		fb_edit_mfps_bestuecken_b.st_config.b_config_fertig := FALSE;
		fb_edit_mfps_bestuecken_b.st_config.b_station_aktiv := TRUE;
		fb_edit_mfps_bestuecken_b.st_config.i16_meld_startindex := 860;
		fb_edit_mfps_bestuecken_b.st_config.str_beschreibung := ' ';
		fb_edit_mfps_bestuecken_b.st_config.str_instanz_name := 'Kurvenscheibeneditor Bestücken B-Achse';
		fb_edit_mfps_bestuecken_b.st_config.b_config_fertig := TRUE;

		fb_camtable_bestueckachse.st_config.b_config_fertig := FALSE;
		fb_camtable_bestueckachse.st_config.b_station_aktiv := TRUE;
		fb_camtable_bestueckachse.st_config.i16_meld_startindex := 880;
		fb_camtable_bestueckachse.st_config.str_beschreibung := ' ';
		fb_camtable_bestueckachse.st_config.str_instanz_name := 'Kurvenscheibeneditor Bestückachse';
		fb_camtable_bestueckachse.st_config.b_config_fertig := TRUE;

		(* Bestückbildgenerierung *)
		bbgen.st_config.b_config_fertig := FALSE;
		bbgen.st_config.b_station_aktiv := TRUE;
		bbgen.st_config.i16_meld_startindex := 700;
		bbgen.st_config.str_beschreibung := ' ';
		bbgen.st_config.str_instanz_name := 'Bestückbildgenerierung';
		bbgen.st_config.b_config_fertig := TRUE;
		
		(* Barcodereader *)
		barcode.fb.st_config.b_config_fertig := FALSE;
		barcode.fb.st_config.b_station_aktiv := TRUE;
		barcode.fb.st_config.i16_meld_startindex := 720;
		barcode.fb.st_config.str_beschreibung := ' ';
		barcode.fb.st_config.str_instanz_name := 'Barcodereader';
		barcode.fb.st_config.b_config_fertig := TRUE;
		
		(* Ballufftagreader *)
		balluff_tag_reader.fb.st_config.b_config_fertig := FALSE;
		balluff_tag_reader.fb.st_config.b_station_aktiv := TRUE;
		balluff_tag_reader.fb.st_config.i16_meld_startindex := 740;
		balluff_tag_reader.fb.st_config.str_beschreibung := ' ';
		balluff_tag_reader.fb.st_config.str_instanz_name := 'Ballufftagreader';
		balluff_tag_reader.fb.st_config.b_config_fertig := TRUE;

		(* WT-Transport Warteposition 1720 *)
		wt_transport_warteposition_1720.st_config.b_config_fertig := FALSE;
		wt_transport_warteposition_1720.st_config.i16_meld_startindex := 760;
		wt_transport_warteposition_1720.st_config.str_beschreibung := ' ';
		wt_transport_warteposition_1720.st_config.str_instanz_name := 'WT-Transport Warteposition 1720';
		wt_transport_warteposition_1720.st_config.b_config_fertig := TRUE;
		
		(* WT-Transport Beladestation 1720 *)
		wt_transport_beladen_1720.st_config.b_config_fertig := FALSE;
		wt_transport_beladen_1720.st_config.i16_meld_startindex := 780;
		wt_transport_beladen_1720.st_config.str_beschreibung := ' ';
		wt_transport_beladen_1720.st_config.str_instanz_name := 'WT-Transport Beladestation 1720';
		wt_transport_beladen_1720.st_config.b_config_fertig := TRUE;
		
		(* Rasterfolienmontge *)
		rasterfolienmontage.st_config.b_config_fertig := FALSE;
		rasterfolienmontage.st_config.b_station_aktiv := TRUE;
		rasterfolienmontage.st_config.i16_meld_startindex := 800;
		rasterfolienmontage.st_config.str_beschreibung := ' ';
		rasterfolienmontage.st_config.str_instanz_name := 'Rasterfolienmontge';
		rasterfolienmontage.st_config.b_config_fertig := TRUE;
		
		(* Rasterfolieneinzug *)
		rasterfolieneinzug.st_config.b_config_fertig := FALSE;
		rasterfolieneinzug.st_config.b_station_aktiv := TRUE;
		rasterfolieneinzug.st_config.i16_meld_startindex := 820;
		rasterfolieneinzug.st_config.str_beschreibung := ' ';
		rasterfolieneinzug.st_config.str_instanz_name := 'Rasterfolieneinzug';
		rasterfolieneinzug.st_config.b_config_fertig := TRUE;

		(*Tag lesen und schreiben *)
		Lesen_Schreiben_Tag.st_config.b_config_fertig := FALSE;
		Lesen_Schreiben_Tag.st_config.b_station_aktiv := TRUE;
		Lesen_Schreiben_Tag.st_config.i16_meld_startindex := 840;
		Lesen_Schreiben_Tag.st_config.str_beschreibung := ' ';
		Lesen_Schreiben_Tag.st_config.str_instanz_name := 'Tag lesen und schreiben';
		Lesen_Schreiben_Tag.st_config.b_config_fertig := TRUE;

		(* Wartung *)
		wartung.st_config.b_config_fertig := FALSE;
		wartung.st_config.b_station_aktiv := TRUE;
		wartung.st_config.i16_meld_startindex := 920;
		wartung.st_config.str_beschreibung := ' ';
		wartung.st_config.str_instanz_name := 'Wartung';
		wartung.st_config.b_config_fertig := TRUE;

		(*Service *)
		Service.st_config.b_config_fertig := FALSE;
		Service.st_config.b_station_aktiv := TRUE;
		Service.st_config.i16_meld_startindex := 900;
		Service.st_config.str_beschreibung := ' ';
		Service.st_config.str_instanz_name := 'Service';
		Service.st_config.b_config_fertig := TRUE;

		(*TouchProbe *)
		ST_TouchProbe.st_config.b_config_fertig := FALSE;
		ST_TouchProbe.st_config.b_station_aktiv := TRUE;
		ST_TouchProbe.st_config.i16_meld_startindex := 940;
		ST_TouchProbe.st_config.str_beschreibung := ' ';
		ST_TouchProbe.st_config.str_instanz_name := 'TouchProbe';
		ST_TouchProbe.st_config.b_config_fertig := TRUE;

		(*AutocheckinDaten *)
		ST_AutoCheckIn.fb_AutocheckinDaten.st_config.b_config_fertig:= FALSE;
		ST_AutoCheckIn.fb_AutocheckinDaten.st_config.b_station_aktiv:= TRUE;
		ST_AutoCheckIn.fb_AutocheckinDaten.st_config.i16_meld_startindex:=	960;
		ST_AutoCheckIn.fb_AutocheckinDaten.st_config.str_beschreibung:= ' ';
		ST_AutoCheckIn.fb_AutocheckinDaten.st_config.str_instanz_name:=	'AutoCheckInDaten';
		ST_AutoCheckIn.fb_AutocheckinDaten.st_config.b_config_fertig:= TRUE;

		(* WT-Transport Warteposition Achse 1700 *)
		wt_transport_warteposition_1700.st_config.b_config_fertig := FALSE;
		wt_transport_warteposition_1700.st_config.i16_meld_startindex := 400;
		wt_transport_warteposition_1700.st_config.str_beschreibung := ' ';
		wt_transport_warteposition_1700.st_config.str_instanz_name := 'WT-Transport Warteposition 1700';
		wt_transport_warteposition_1700.st_config.b_config_fertig := TRUE;
		
		(* WT-Transport Beladestation Achse 1700 *)
		wt_transport_beladen_achse_1700.st_config.b_config_fertig := FALSE;
		wt_transport_beladen_achse_1700.st_config.i16_meld_startindex := 420;
		wt_transport_beladen_achse_1700.st_config.str_beschreibung := ' ';
		wt_transport_beladen_achse_1700.st_config.str_instanz_name := 'WT-Transport Beladestation Achse 1700';
		wt_transport_beladen_achse_1700.st_config.b_config_fertig := TRUE;

		(* EtherCAT Diagnose *)
		Index:=1;
		EtherCatDiag[Index].st_config.b_config_fertig := FALSE;
		EtherCatDiag[Index].st_config.b_station_aktiv := TRUE;
		EtherCatDiag[Index].st_config.i16_meld_startindex := 980;
		EtherCatDiag[Index].st_config.str_beschreibung := ' ';
		EtherCatDiag[Index].st_config.str_instanz_name := 'Grundmaschine';
		EtherCatDiag[Index].st_config.b_config_fertig := TRUE;

		(* EtherCAT Diagnose *)
		Index:=2;
		EtherCatDiag[Index].st_config.b_config_fertig := FALSE;
		EtherCatDiag[Index].st_config.b_station_aktiv := TRUE;
		EtherCatDiag[Index].st_config.i16_meld_startindex := 985;
		EtherCatDiag[Index].st_config.str_beschreibung := ' ';
		EtherCatDiag[Index].st_config.str_instanz_name := 'Hublift links';
		EtherCatDiag[Index].st_config.b_config_fertig := TRUE;

		(* EtherCAT Diagnose *)
		Index:=3;
		EtherCatDiag[Index].st_config.b_config_fertig := FALSE;
		EtherCatDiag[Index].st_config.b_station_aktiv := TRUE;
		EtherCatDiag[Index].st_config.i16_meld_startindex := 990;
		EtherCatDiag[Index].st_config.str_beschreibung := ' ';
		EtherCatDiag[Index].st_config.str_instanz_name := 'Hublift rechts';
		EtherCatDiag[Index].st_config.b_config_fertig := TRUE;

		(* EtherCAT Diagnose *)
		Index:=4;
		EtherCatDiag[Index].st_config.b_config_fertig := FALSE;
		EtherCatDiag[Index].st_config.b_station_aktiv := TRUE;
		EtherCatDiag[Index].st_config.i16_meld_startindex := 995;
		EtherCatDiag[Index].st_config.str_beschreibung := ' ';
		EtherCatDiag[Index].st_config.str_instanz_name := 'Bandeinzug';
		EtherCatDiag[Index].st_config.b_config_fertig := TRUE;

		(* Melde-Arrays rücksetzen *)
		FOR i := 0 TO SIZEOF (garr_stoermeldungen) / SIZEOF (garr_stoermeldungen[0]) - 1 BY 1 DO
			garr_stoermeldungen[i] := 0;
		END_FOR
		FOR i := 0 TO SIZEOF (garr_betriebsmeldungen) / SIZEOF (garr_betriebsmeldungen[0]) - 1 BY 1 DO
			garr_betriebsmeldungen[i] := 0;
		END_FOR
ELSE
	b_config_fertig := TRUE;
END_IF

		
		
END_PROGRAM

(* POU Gemeinsamkeiten17xx/Achsen/ST_TouchProbe, ST *)
PROGRAM ST_TouchProbe
VAR_INPUT
	st_config						: struct_config;
	st_ctrl_in						: struct_ctrl_in;
END_VAR
VAR_OUTPUT
	st_ctrl_out					: struct_ctrl_out;
END_VAR
VAR
	fb_state_entry				: ST_StateEntry;
	st_ctrl_in_empty				: struct_ctrl_in;
	fb_ton_quitt					: TON;
	fb_ton_uez					: TON;
	fb_ton_wz					: TON;

	sm_CompareY				:BOOL;
	sm_CompareZ				:BOOL;
	sm_keinMessergebnisY		:BOOL;
	sm_keinMessergebnisZ		:BOOL;
	sm_WtAufSchlitten				:BOOL;

	i16_Counter					:INT;

	fb_TouchProbeLog			: FB_ExporString;	(* Fehlermeldungen in Errorlog (txt) schreiben *)
	s_FileName					: STRING;			(* Name Errorlogdatei *)
	s_ExportStr					: T_MaxString;		(* kompletter Text zum Eintrag in Errorlog *)
	s_ProductionsDate				: STRING;		(* Datum für Logeintrag *)

	lr_RecPosZ					:LREAL;		(*Wird beim Anlagenstart beschrieben*)
	lr_RecPosY					:LREAL;		(*Wird beim Anlagenstart beschrieben*)

END_VAR

VAR CONSTANT
	Trennzeichen					: STRING(3):=' |';
END_VAR
(*======================================================
   PRG: ST_TouchProbe
 ------------------------------------------------------
   Auth: 		Werner Friedl    						 
   Date: 		10.09.2019    						     
   Rev.: 		1.0	
   Desc:		Es werden nacheinander die Z- und Y Achse auf einen Messtaster gefahren und dabei
			die Ermittelten Tastpositionen in ein Lofile eingetregen. ("Projektpad"\TouchProbeLog)

			ACHTUNG!		auf dem Schlitten darf kein WT sein
							bei allen Anlagen Softwarelimits überprüfen und die Taster so motieren, dass sie kurz vor dem Softwarelimit schalten.

			Ablauf und Funktion.
			- bei einem Anlagen Neustart wird das erste Messergebnis in die VAR lr_RecPosZ und lr_RecPosY eingetragen.
			  Diese Messwerte werden dann mit allen darauf folgenden Messungen verglichen.
			- im Prg. "ST_AxisJobCtrl_Motion" muss die Touchprobe Funktion eingefügt sein ( MOVE_TOUCH_PROBE)

			gst_datensatz.st_md.lr_ToleranzTouchProbe				(Toleranz für den Vergleich)
			gst_datensatz.st_md.i16_WdhTouchProbe				(Anzahl der WT-wechsel bis zur nächsten Messung bei 0 wird keine Prüfung gemacht)

			Das Programm wird im ST_WT_Transport_Beladen gestartet (Schritt 140)

   Historie:   1.0

 ========================================================*)
(* Zeiten *)
fb_ton_wz(IN:= , PT:= , Q=>  , ET=> );
fb_ton_uez(IN:= , PT:= , Q=>  , ET=> );
fb_ton_quitt(IN:= , PT:= t#100ms, Q=> , ET=> );

(* Flanken *)

(* Toplevel *)
IF fb_state_entry.i16_next_step > INIT AND fb_state_entry.i16_next_step < FEHLER THEN
	IF fb_state_entry.i16_next_step < STOP THEN
		IF st_ctrl_in.b_stop THEN
			fb_state_entry.i16_next_step := STOP;
		END_IF
	END_IF

	IF	axis_y_achse.st_ctrl.out.b_fehler	OR
		axis_z_achse.st_ctrl.out.b_fehler OR
		NOT ST_Safetyprogramm.se_steuerung_ein THEN
		fb_state_entry.i16_next_step := FEHLER;
	END_IF

END_IF

(* ==================================Schrittkette================================ *)
fb_state_entry(i16_pos:= 1);

CASE fb_state_entry.i16_step OF
(*=======================================================*)
INIT_OBJ:
	IF st_config.b_config_fertig THEN
		fb_state_entry.i16_next_step := INIT;
	END_IF

(*=======================================================*)
INIT:
	IF fb_state_entry.E THEN
		fb_ton_wz.IN := FALSE;
		fb_ton_uez.IN	:= FALSE;
		fb_ton_quitt.IN := FALSE;

		sm_CompareY:=FALSE;
		sm_CompareZ:=FALSE;
		sm_keinMessergebnisY:=FALSE;
		sm_keinMessergebnisZ:=FALSE;
		sm_WtAufSchlitten:=	FALSE;
	END_IF

	(*-----------------------Weiterschaltbedingungen----------------------------*)
	IF 	st_ctrl_in.b_init THEN
		fb_state_entry.i16_next_step := 20;
	END_IF

(*=======================================================*)
20: (* Initialisierung*)

	(*-----------------------Weiterschaltbedingungen----------------------------*)
	fb_state_entry.i16_next_step := BEREIT;

(*=======================================================*)
BEREIT:	(* Warte auf Anforderung von vorheriger Station zum aufnehmen des WT *)
	IF 	fb_state_entry.E THEN
		st_ctrl_out.b_bereit := TRUE;
	END_IF

	(*-----------------------Weiterschaltbedingungen----------------------------*)
	IF 	st_ctrl_in.b_start  OR st_ctrl_in.b_start_2 THEN
		fb_state_entry.i16_next_step := 110;
	END_IF

	IF 	fb_state_entry.X THEN
		st_ctrl_out.b_fertig := FALSE;
		st_ctrl_out.b_busy := TRUE;
	END_IF

(*=======================================================*)
110: (* Prüfe Startbedinung*)

	(*-----------------------Weiterschaltbedingungen----------------------------*)
	(*Prüfen ob ein Taster angeklemmt ist*)
	IF	NOT ST_Z_Achse.fb_axis.b_TriggerInput OR
		gst_datensatz.st_md.i16_WdhTouchProbe <= 0 OR
		gst_datensatz.st_md.lr_ToleranzTouchProbe <= 0 THEN
		fb_state_entry.i16_next_step := BEREIT;
		st_ctrl_out.b_fertig := TRUE;
		st_ctrl_out.b_busy := FALSE;
	ELSE
		IF	i16_Counter >= gst_datensatz.st_md.i16_WdhTouchProbe  OR
			i16_Counter = 0 THEN
			fb_state_entry.i16_next_step := 115;
		ELSE
			st_ctrl_out.b_fertig := TRUE;
			st_ctrl_out.b_busy := FALSE;
			fb_state_entry.i16_next_step := BEREIT;
		END_IF
	END_IF

	IF 	fb_state_entry.X THEN
		i16_Counter:=i16_Counter+1;
	END_IF

(*=======================================================*)
115: (* Prüfe ob Schlitten ohne WT ist*)
	IF fb_state_entry.E THEN
		fb_ton_wz.PT := t#1000ms;
	END_IF

	IF	gst_datensatz.st_md.i16_typ_zelle = BESTUECKZELLE_1720   THEN
		fb_ton_wz.IN:=ST_WT_Transport_Beladen_1720.e_wt_auf_beladepos;
		IF NOT ST_WT_Transport_Beladen_1720.e_wt_auf_beladepos THEN
			fb_state_entry.i16_next_step := 120;
		END_IF
	ELSE
		fb_ton_wz.IN:=ST_WT_Transport_Beladen.e_wt_auf_beladepos;
		IF NOT ST_WT_Transport_Beladen.e_wt_auf_beladepos THEN
			fb_state_entry.i16_next_step := 120;
		END_IF
	END_IF

	IF	fb_ton_wz.Q THEN
		sm_WtAufSchlitten:=TRUE;
		fb_state_entry.i16_next_step := FEHLER;
	END_IF

	IF fb_state_entry.X THEN
		fb_ton_wz.IN := FALSE;
	END_IF

(*=======================================================*)
120: (* CAM_OUT_SLAVE*)
	IF fb_state_entry.E THEN
		ST_Z_Achse.b_start_in := TRUE;
	END_IF

	(*-----------------------Weiterschaltbedingungen----------------------------*)
	IF	axis_z_achse.st_ctrl.out.b_busy  THEN
		fb_state_entry.i16_next_step := 122;
	END_IF

(*=======================================================*)
122:(*warten auf  fertig*)
	(*-----------------------Weiterschaltbedingungen----------------------------*)
	IF	axis_z_achse.st_ctrl.out.b_fertig  THEN
		fb_state_entry.i16_next_step := 124;
	END_IF

(*=======================================================*)
124:(*prüfe CoupleState*)

	IF 	(y_achse.NcToPlc.CoupleState = 0 OR gst_datensatz.st_md.i16_typ_zelle = BESTUECKZELLE_1720)AND
	 	z_achse.NcToPlc.CoupleState = 0  THEN
		fb_state_entry.i16_next_step := 126;
	END_IF

(*=======================================================*)
126: (* Z-Achse vor TouchProbe fahren*)
	IF fb_state_entry.E THEN
		ST_Z_Achse.lr_Achspos_in:=-95 + 20 ;				(*Taster befindet sich in Der Nähe vom Motor*)
		ST_Z_Achse.lr_Velo_in:=ST_Z_Achse.st_geschwindigkeiten.lr_auto_max ;
		ST_Z_Achse.enu_cmd_in:=MOVE_TOUCH_PROBE;
		ST_Z_Achse.b_start_in := TRUE;
	END_IF

	(*-----------------------Weiterschaltbedingungen----------------------------*)
	IF	axis_z_achse.st_ctrl.out.b_busy  THEN
		fb_state_entry.i16_next_step := 128;
	END_IF

(*=======================================================*)
128:(*warten auf  fertig*)
	(*-----------------------Weiterschaltbedingungen----------------------------*)
	IF	axis_z_achse.st_ctrl.out.b_fertig  THEN
		fb_state_entry.i16_next_step := 130;
	END_IF

(*=======================================================*)
130: (* Z-Achse auf TouchProbe fahren*)
	IF fb_state_entry.E THEN
		ST_Z_Achse.lr_Achspos_in:=-95 ;				(*Taster befindet sich in Der Nähe vom Motor*)
		ST_Z_Achse.lr_Velo_in:=ST_Z_Achse.st_geschwindigkeiten.lr_auto_max / 5;
		ST_Z_Achse.enu_cmd_in:=MOVE_TOUCH_PROBE;
		ST_Z_Achse.b_start_in := TRUE;
	END_IF

	(*-----------------------Weiterschaltbedingungen----------------------------*)
	IF	axis_z_achse.st_ctrl.out.b_busy  THEN
		fb_state_entry.i16_next_step := 132;
	END_IF

(*=======================================================*)
132:(*warten auf  fertig*)
	(*-----------------------Weiterschaltbedingungen----------------------------*)
	IF	axis_z_achse.st_ctrl.out.b_fertig  THEN
		fb_state_entry.i16_next_step := 134;
	END_IF

(*=======================================================*)
134: (* Z-Achse vom TouchProbe runter fahren und Positionieren für die Y Achse *)
	IF fb_state_entry.E THEN
		IF	gst_datensatz.st_md.i16_typ_zelle <> BESTUECKZELLE_1720 THEN
			ST_Z_Achse.lr_Achspos_in:=70;				(*Taster befindet sich in DerNähe vom Motor*)
		ELSE
			ST_Z_Achse.lr_Achspos_in:=gst_datensatz.st_md.st_md_z_achse.lr_wt_uebergabepos  ;
		END_IF
		ST_Z_Achse.lr_Velo_in:=ST_Z_Achse.st_geschwindigkeiten.lr_auto_max ;
		ST_Z_Achse.enu_cmd_in:=MOVE_ABSOLUTE;
		ST_Z_Achse.b_start_in := TRUE;
	END_IF

	(*-----------------------Weiterschaltbedingungen----------------------------*)
	IF	axis_z_achse.st_ctrl.out.b_busy  THEN
		fb_state_entry.i16_next_step := 140;
	END_IF

(*=======================================================*)
140:(*warten auf  fertig*)
	(*-----------------------Weiterschaltbedingungen----------------------------*)
	IF	axis_z_achse.st_ctrl.out.b_fertig  THEN

		IF	gst_datensatz.st_md.i16_typ_zelle = BESTUECKZELLE_1720 THEN
			fb_state_entry.i16_next_step := 220;
		ELSE
			fb_state_entry.i16_next_step := 150;
		END_IF
	END_IF

(*=======================================================*)
150: (* Y-Achse auf TouchProbe fahren*)
	IF fb_state_entry.E THEN
		ST_Y_Achse.lr_Achspos_in:=30;				(*Taster befindet sich in der Nähe vom Motor*)
		ST_Y_Achse.lr_Velo_in:=ST_Y_Achse.st_geschwindigkeiten.lr_auto_max;
		ST_Y_Achse.enu_cmd_in:=MOVE_ABSOLUTE;
		ST_Y_Achse.b_start_in := TRUE;
	END_IF

	(*-----------------------Weiterschaltbedingungen----------------------------*)
	IF	axis_y_achse.st_ctrl.out.b_busy  THEN
		fb_state_entry.i16_next_step := 160;
	END_IF

(*=======================================================*)
160:(*warten auf  fertig*)
	(*-----------------------Weiterschaltbedingungen----------------------------*)
	IF	axis_y_achse.st_ctrl.out.b_fertig  THEN
		fb_state_entry.i16_next_step := 162;
	END_IF

(*=======================================================*)
162: (* Y-Achse auf TouchProbe fahren*)
	IF fb_state_entry.E THEN
		ST_Y_Achse.lr_Achspos_in:=65;				(*Taster befindet sich in der Nähe vom Motor*)
		ST_Y_Achse.lr_Velo_in:=ST_Y_Achse.st_geschwindigkeiten.lr_auto_max / 5;
		ST_Y_Achse.enu_cmd_in:=MOVE_TOUCH_PROBE;
		ST_Y_Achse.b_start_in := TRUE;
	END_IF

	(*-----------------------Weiterschaltbedingungen----------------------------*)
	IF	axis_y_achse.st_ctrl.out.b_busy  THEN
		fb_state_entry.i16_next_step := 164;
	END_IF

(*=======================================================*)
164:(*warten auf  fertig*)
	(*-----------------------Weiterschaltbedingungen----------------------------*)
	IF	axis_y_achse.st_ctrl.out.b_fertig  THEN
		fb_state_entry.i16_next_step := 170;
	END_IF

(*=======================================================*)
170: (* Y-Achse vom TouchProbe runter fahren*)
	IF fb_state_entry.E THEN
		ST_Y_Achse.lr_Achspos_in:=30 ;
		ST_Y_Achse.lr_Velo_in:=ST_Y_Achse.st_geschwindigkeiten.lr_auto_max;
		ST_Y_Achse.enu_cmd_in:=MOVE_ABSOLUTE;
		ST_Y_Achse.b_start_in := TRUE;
	END_IF

	(*-----------------------Weiterschaltbedingungen----------------------------*)
	IF	axis_y_achse.st_ctrl.out.b_busy  THEN
		fb_state_entry.i16_next_step := 180;
	END_IF

(*=======================================================*)
180:(*warten auf  Vorschub zurück fertig*)
	(*-----------------------Weiterschaltbedingungen----------------------------*)
	IF	axis_y_achse.st_ctrl.out.b_fertig  THEN
		fb_state_entry.i16_next_step := 190;
	END_IF

(*=======================================================*)
190: (* Y-Achse vom TouchProbe runter fahren*)
	IF fb_state_entry.E THEN
		ST_Y_Achse.lr_Achspos_in:=gst_datensatz.st_md.st_md_y_achse.lr_wt_uebergabepos;
		ST_Y_Achse.enu_cmd_in:=MOVE_ABSOLUTE;
		ST_Y_Achse.b_start_in := TRUE;
		ST_Z_Achse.lr_Achspos_in:=gst_datensatz.st_md.st_md_z_achse.lr_wt_uebergabepos  ;
		ST_Z_Achse.enu_cmd_in:=MOVE_ABSOLUTE;
		ST_Z_Achse.b_start_in := TRUE;
	END_IF

	(*-----------------------Weiterschaltbedingungen----------------------------*)
	IF	axis_y_achse.st_ctrl.out.b_busy  AND
		axis_z_achse.st_ctrl.out.b_busy THEN
		fb_state_entry.i16_next_step := 200;
	END_IF

(*=======================================================*)
200:(*warten auf  Vorschub zurück fertig*)
	(*-----------------------Weiterschaltbedingungen----------------------------*)
	IF	axis_y_achse.st_ctrl.out.b_fertig AND
		axis_z_achse.st_ctrl.out.b_fertig THEN
		fb_state_entry.i16_next_step := 210;
	END_IF

(*=======================================================*)
210: (* Y- und Z_Achse auf Startposition fahren*)
	IF fb_state_entry.E THEN
		ST_Z_Achse.enu_cmd_in:=CAM_IN_SLAVE;			(*Y-Achse wird wieder angekoppelt*)
		ST_Z_Achse.b_start_in := TRUE;
	END_IF

	(*-----------------------Weiterschaltbedingungen----------------------------*)
	IF	axis_z_achse.st_ctrl.out.b_busy THEN
		fb_state_entry.i16_next_step := 220;
	END_IF

(*=======================================================*)
220:(*warten auf  Vorschub zurück fertig*)
	(*-----------------------Weiterschaltbedingungen----------------------------*)
	IF	axis_z_achse.st_ctrl.out.b_fertig  THEN
		fb_state_entry.i16_next_step := 230;
		st_ctrl_out.b_fertig := TRUE;
		st_ctrl_out.b_busy := FALSE;
	END_IF

(*=======================================================*)
230:(*Wenn die RecPos=0 sind dann funktionieren die Messtaster nicht*)

	IF	gst_datensatz.st_md.i16_typ_zelle <> BESTUECKZELLE_1720 THEN
		sm_keinMessergebnisY := ST_Y_Achse.lr_RecPos = 0;
	END_IF
	sm_keinMessergebnisZ := ST_Z_Achse.lr_RecPos = 0;

	(*-----------------------Weiterschaltbedingungen----------------------------*)
	IF	sm_keinMessergebnisY OR
		sm_keinMessergebnisZ THEN
		fb_state_entry.i16_next_step := FEHLER;
	ELSE
		fb_state_entry.i16_next_step := 500;
		i16_Counter:=1;
	END_IF

(*=======================================================*)
500:	(*Eintrag in die ErrorLog===========================================*)
	IF	fb_state_entry.E THEN

		s_ProductionsDate:=DT_TO_SPECIALSTRING_YYYY_MM(inDT:=gdt_system_time);
		s_FileName:=CONCAT('TouchProbeLog_',s_ProductionsDate);
		s_FileName:=CONCAT(s_FileName,'.txt');
		s_ExportStr:=DELETE(DT_TO_STRING(gdt_system_time),3,1);
		s_ExportStr:=CONCAT(s_ExportStr,Trennzeichen);
		s_ExportStr:=CONCAT(s_ExportStr,'Axis Z: ');
		s_ExportStr:=CONCAT(s_ExportStr,LREAL_TO_FMTSTR(ST_Z_Achse.lr_RecPos,5,TRUE));
		IF	gst_datensatz.st_md.i16_typ_zelle <> BESTUECKZELLE_1720 THEN
			s_ExportStr:=CONCAT(s_ExportStr,Trennzeichen);
			s_ExportStr:=CONCAT(s_ExportStr,'Axis Y: ');
			s_ExportStr:=CONCAT(s_ExportStr,LREAL_TO_FMTSTR(ST_Y_Achse.lr_RecPos,5,TRUE));
		END_IF

		IF 	lr_RecPosY = 0 THEN		(*Wird beim Anlagenstart beschrieben*)
			lr_RecPosY:= ST_Y_Achse.lr_RecPos;
		END_IF

		IF 	lr_RecPosZ = 0 THEN		(*Wird beim Anlagenstart beschrieben*)
			lr_RecPosZ:= ST_Z_Achse.lr_RecPos;
			s_ExportStr:=CONCAT(s_ExportStr,' start compare ');
		END_IF

		sm_CompareY:=ABS(lr_RecPosY - ST_Y_Achse.lr_RecPos) > gst_datensatz.st_md.lr_ToleranzTouchProbe;
		sm_CompareZ:=ABS(lr_RecPosZ - ST_Z_Achse.lr_RecPos) > gst_datensatz.st_md.lr_ToleranzTouchProbe;

		IF 	sm_CompareY OR
			sm_CompareZ THEN
			s_ExportStr:=CONCAT(s_ExportStr,' error compare   difference > ');
			s_ExportStr:=CONCAT(s_ExportStr,LREAL_TO_FMTSTR(gst_datensatz.st_md.lr_ToleranzTouchProbe,4,TRUE));
		END_IF

	END_IF

	(*-----------------------Weiterschaltbedingungen----------------------------*)
	IF	NOT fb_TouchProbeLog.Busy AND
		NOT fb_TouchProbeLog.Error  THEN
		fb_state_entry.i16_next_step:=510;
	ELSE
		fb_state_entry.i16_next_step:=FEHLER;
	END_IF

(*=======================================================*)
510:	(* Starte Schreibvorgang *)
	IF	fb_state_entry.E THEN
		fb_TouchProbeLog.Start:=TRUE;
	END_IF

	(*-----------------------Weiterschaltbedingungen----------------------------*)
	IF	NOT fb_TouchProbeLog.Busy AND
		fb_TouchProbeLog.Done THEN
		fb_state_entry.i16_next_step:=BEREIT;
	END_IF
	IF	fb_TouchProbeLog.Error OR
		sm_CompareY OR
 		sm_CompareZ THEN
		fb_state_entry.i16_next_step:=FEHLER;
	END_IF


(*=======================================================*)
FEHLER:
	IF fb_state_entry.E THEN
		fb_ton_quitt.IN := FALSE;
		st_ctrl_out.b_fehler := TRUE;
		st_ctrl_out.b_bereit := FALSE;
		st_ctrl_out.b_fertig := FALSE;
		st_ctrl_out.b_busy := FALSE;
	END_IF

	(*-----------------------Weiterschaltbedingungen----------------------------*)
	IF st_ctrl_in.b_quitt AND NOT fb_state_entry.E THEN
		st_ctrl_out.b_fehler := FALSE;
		fb_ton_quitt.IN := TRUE;
	END_IF


	IF fb_ton_quitt.Q THEN
		fb_ton_quitt.IN := FALSE;
		fb_state_entry.i16_next_step := INIT;
	END_IF

(*=======================================================*)
STOP:
	IF fb_state_entry.E THEN
		fb_ton_quitt.IN := FALSE;
		st_ctrl_out.b_gestoppt := TRUE;
		st_ctrl_out.b_bereit := FALSE;
		st_ctrl_out.b_fertig := FALSE;
		st_ctrl_out.b_busy := FALSE;
	END_IF

	(*-----------------------Weiterschaltbedingungen----------------------------*)
	IF 	st_ctrl_in.b_quitt AND NOT fb_state_entry.E THEN
		st_ctrl_out.b_gestoppt := FALSE;
		fb_ton_quitt.IN := TRUE;
	END_IF

	IF fb_ton_quitt.Q THEN
		fb_ton_quitt.IN := FALSE;
		fb_state_entry.i16_next_step := INIT;
	END_IF
END_CASE

st_ctrl_in:=st_ctrl_in_empty;

fb_state_entry(i16_pos:= 2);

IF st_config.b_config_fertig THEN
	(* Fehlermeldungen und Betriebsmeldungen ab dem Startindex in die globalen Meldungsarrays schreiben *)
	garr_stoermeldungen[st_config.i16_meld_startindex + 0] := sm_CompareY;
	garr_stoermeldungen[st_config.i16_meld_startindex + 1] := sm_CompareZ;
	garr_stoermeldungen[st_config.i16_meld_startindex + 2] := sm_keinMessergebnisY;
	garr_stoermeldungen[st_config.i16_meld_startindex + 3] := sm_keinMessergebnisZ;
	garr_stoermeldungen[st_config.i16_meld_startindex + 4] := sm_WtAufSchlitten;
	garr_stoermeldungen[st_config.i16_meld_startindex + 5] := FALSE;
	garr_stoermeldungen[st_config.i16_meld_startindex + 6] := FALSE;
	garr_stoermeldungen[st_config.i16_meld_startindex + 7] := FALSE;
	garr_stoermeldungen[st_config.i16_meld_startindex + 8] := FALSE;
	garr_stoermeldungen[st_config.i16_meld_startindex + 9] := FALSE;

	garr_betriebsmeldungen[st_config.i16_meld_startindex + 0] := FALSE;
	garr_betriebsmeldungen[st_config.i16_meld_startindex + 1] := FALSE;
	garr_betriebsmeldungen[st_config.i16_meld_startindex + 2] := FALSE;
	garr_betriebsmeldungen[st_config.i16_meld_startindex + 3] := FALSE;
	garr_betriebsmeldungen[st_config.i16_meld_startindex + 4] := FALSE;
	garr_betriebsmeldungen[st_config.i16_meld_startindex + 5] := FALSE;
	garr_betriebsmeldungen[st_config.i16_meld_startindex + 6] := FALSE;
	garr_betriebsmeldungen[st_config.i16_meld_startindex + 7] := FALSE;
	garr_betriebsmeldungen[st_config.i16_meld_startindex + 8] := FALSE;
	garr_betriebsmeldungen[st_config.i16_meld_startindex + 9] := FALSE;

END_IF


fb_TouchProbeLog(
	Start:= ,
	Reset:= ,
	ExportStr:= s_ExportStr,
	FileName:= s_FileName,
	Path:=  CONCAT(s_Projekt_path,'TouchProbeLog\'),
	Mode:=FOPEN_MODEAPPEND,	(*am Ende anhängen*)
	Ready=> ,
	Busy=> ,
	Done=> ,
	Error=> ,
	ErrorMsg=> );
END_PROGRAM

(* POU EPT Lib/Daten/FB_ExporString, ST *)
FUNCTION_BLOCK FB_ExporString
VAR_INPUT
	Start				:BOOL;
	Reset			:BOOL;
	ExportStr			:STRING(255);
	FileName		:STRING(255);
	Path				:STRING(255);
	Mode			:DWORD;
END_VAR
VAR_OUTPUT
	Ready				:BOOL;
	Busy				:BOOL;
	Done				:BOOL;
	Error				:BOOL;
	ErrorMsg			:STRING(255);

END_VAR
VAR
	fb_state_entry		:ST_StateEntry;
	nErrId				:UDINT;
	i					:UINT;

	fbFileOpen			:FB_FileOpen;
	fbFilePuts			:FB_FilePuts;
	fbFileClose			:FB_FileClose;

	hFile				:UINT;

	ProductionDate		:STRING;

END_VAR

VAR CONSTANT
	Zeilenumbruch		:STRING:='$R$N';
END_VAR
(*======================================================
   PRG: FB_ExportString
 ------------------------------------------------------
   Auth: 		Werner Friedl    						 
   Date: 		30.10.2014    						     
   Rev.: 		1.0	
   Desc:		
		
   Historie:   1.0

 ========================================================*)
fb_state_entry(i16_pos:= 1);

CASE fb_state_entry.i16_step OF

0:	(*Objekt initialisieren*)
	fb_state_entry.i16_next_step:=INIT;

10:	(*initialisieren*)
	fb_state_entry.i16_next_step:=BEREIT;

BEREIT:(*Start*)

	IF	Start THEN  (*initialisieren*)
		Start:=FALSE;
		Busy:=TRUE;
		Error:=FALSE;
		Done:=FALSE;
		nErrId:=0;
		ErrorMsg:='';
		fb_state_entry.i16_next_step:=110;

	END_IF

110: (*Datei erstellen*)

	FileName:=CONCAT(Path,FileName);

	fbFileOpen.sPathName:=FileName;
 	fbFileOpen.bExecute:=TRUE;

	IF 	NOT fbFileOpen.bBusy   THEN
		fb_state_entry.i16_next_step:=120;
	END_IF

120: (*Datei erstellen*)

	IF 	NOT fbFileOpen.bBusy THEN
		fbFileOpen.bExecute:=FALSE;
		IF 	fbFileOpen.bError THEN
			nErrId:=fbFileOpen.nErrId;
			fb_state_entry.i16_next_step:=FEHLER;
			ErrorMsg:='Fehler beim Öffnen der Datei';
		ELSE
			fb_state_entry.i16_next_step:=130;
		END_IF
	END_IF

130: (*String in Datei eintragen*)
	IF fb_state_entry.E THEN
		;
	END_IF

	fbFilePuts.sLine:=CONCAT(ExportStr,Zeilenumbruch);
	fbFilePuts.bExecute:=TRUE;

	IF  fbFilePuts.bBusy THEN
		fb_state_entry.i16_next_step:=140;
	END_IF

140: (*String in Datei eintragen*)

	IF 	NOT fbFilePuts.bBusy THEN
		fbFilePuts.bExecute:=FALSE;
		IF 	fbFilePuts.bError THEN
			nErrId:=fbFilePuts.nErrId;
			fb_state_entry.i16_next_step:=150;
			ErrorMsg:='Fehler beim String Eintragen in der Datei';
			Error:=TRUE;
		ELSE
			fb_state_entry.i16_next_step:=150;
		END_IF
	END_IF

150:(*Datei schließen*)

	fbFileClose.bExecute:=TRUE;
	IF 	fbFileClose.bBusy THEN
		fb_state_entry.i16_next_step:=160;
	END_IF

160:(*Datei schließen*)

	IF NOT fbFileClose.bBusy THEN
		fbFileClose.bExecute:=FALSE;
		IF 	fbFileClose.bError THEN
			nErrId:=fbFileClose.nErrId;
			ErrorMsg:='Fehler beim Schließen der Datei';
			Error:=TRUE;
		ELSE
			fb_state_entry.i16_next_step:=170;
		END_IF
	END_IF

	IF	Error THEN
		fb_state_entry.i16_next_step:=FEHLER;
	END_IF

170: (*fertig*)
	Busy:=FALSE;
	Done:=TRUE;
	fb_state_entry.i16_next_step:=10;

FEHLER: (*Fehler*)
	fb_state_entry.i16_next_step:=10;
	Busy:=FALSE;
	Error:=TRUE;
END_CASE

fb_state_entry(i16_pos:= 2 );

fbFileOpen(
	sNetId:='',
	sPathName:= ,
	nMode:=mode,
	ePath:=PATH_GENERIC,
	bExecute:= ,
	tTimeout:=T#1s,
	hFile=> hFile);

fbFilePuts(
	sNetId:='',
	hFile:=hFile,
	sLine:= ,
	bExecute:= ,
	tTimeout:=t#1s);

fbFileClose(
	sNetId:='',
	hFile:=hFile,
	bExecute:= ,
	tTimeout:=t#1s);
END_FUNCTION_BLOCK

(* POU Maschine1720/WT Transport/ST_WT_Transport_Beladen_1720, ST *)
PROGRAM ST_WT_Transport_Beladen_1720
VAR_INPUT
	st_config								: struct_config;
	st_ctrl_in								: struct_ctrl_in;
END_VAR
VAR_IN_OUT
	st_visu								: struct_visu;
END_VAR
VAR_OUTPUT
	st_ctrl_out							: struct_ctrl_out;
	t_WT_WechselZeit					: TIME := t#0ms;
	t_traegerwechselzeit					: TIME := t#0ms;
	t_Zentrierer_ausfahren					: TIME := t#0ms;
	t_Zentrierer_einfahren					: TIME := t#0ms;
	t_komplett_zyklus						: TIME := t#0ms;
END_VAR
VAR
	fb_ton_uez							: TON;
	fb_ton_wz							: TON;
	fb_ton_quitt							: TON;
	fb_ton_wt_auf_beladepos				: TON;
	fb_tof_wt_auf_beladepos				: TOF;
	fb_r_trig_start							: R_TRIG;
	fb_r_trig_beladepos					: R_TRIG;
	fb_r_trig_beladepos_verlassen			: R_TRIG;
	fb_state_entry							: ST_StateEntry;
	fb_traegerwechselzeit					: ST_Taktzeit;
	fb_WT_WechselZeit					: ST_Taktzeit;
	fb_Zentrierer_ausfahren				: ST_Taktzeit;
	fb_Zentrierer_einfahren					: ST_Taktzeit;
	t_bestueckzeit						: TIME := t#0ms;
	sm_wt_hat_beladepos_nicht_verlassen	: BOOL := FALSE;
	sm_tagnummer_ungueltig				: BOOL := FALSE;
	sm_wt_hat_kein_tag					: BOOL := FALSE;
	sm_tagreader_nicht_fertig				: BOOL := FALSE;
	sm_keine_bandfreigabe				: BOOL := FALSE;
	bm_abfrage_wt_auf_beladepos			: BOOL := FALSE;
	bm_warte_auf_wt_an_stopper			: BOOL := FALSE;
	bMerkerSchrittketteKommtVonInit		: BOOL := FALSE;
	fb_ton_abfrage_wt_auf_beladepos		: TON;
	fb_ton_warte_auf_wt_an_stopper			: TON;
	i									: INT := 0;

	(* zum Testen der Achsen nach Tausch, Bestückbild "Becherspucken", WKZ ausgebaut, Vorschubkontrolle abeschaltet,
	Bit muss von Programmierer geforct werden, zum Beenden Schlüsselschalter auf HAND und Zelle neu starten *)
	b_Dauertest_Achsen					: BOOL := FALSE;

	e_wt_auf_beladepos					AT %I* : BOOL;
	e_wt_im_aktionsfeld					AT %I* : BOOL;
	e_wt_beladepos_verlassen				AT %I* : BOOL;
	e_wt_auf_pufferstrecke					AT %I* : BOOL;
END_VAR
(* Zeiten *)
fb_ton_uez(IN:= , PT:= , Q=>  , ET=> );
fb_ton_wz(IN:= , PT:= , Q=> , ET=> );
fb_ton_quitt(IN:= , PT:= t#100ms, Q=> , ET=> );

fb_ton_wt_auf_beladepos(IN:= e_wt_auf_beladepos, PT:= t#200ms, Q=> , ET=> );
fb_tof_wt_auf_beladepos(IN:= e_wt_auf_beladepos, PT:= t#200ms, Q=> , ET=> );

(* Flanken *)
fb_r_trig_beladepos(CLK:= e_wt_auf_beladepos, Q=> );
fb_r_trig_beladepos_verlassen(CLK:= e_wt_beladepos_verlassen, Q=> );
fb_r_trig_start(CLK:= st_ctrl_in.b_start, Q=> );

(*Trägerwechselzeiten*)
fb_WT_WechselZeit(b_start:= , t_zeit=> );
fb_Zentrierer_ausfahren(b_start:= , t_zeit=> );
fb_Zentrierer_einfahren(b_start:= , t_zeit=> );


(* ==================================Toplevel=================================== *)
IF fb_state_entry.i16_next_step > INIT AND fb_state_entry.i16_next_step < FEHLER THEN
	(* Allgemeine Fehler *)
	IF st_ctrl_in.b_stop THEN
		fb_state_entry.i16_next_step := STOP;
	ELSIF zyl_wt_zentrierer_tisch.st_ctrl.out.b_fehler OR zyl_wt_stopper_tisch.st_ctrl.out.b_fehler THEN
		fb_state_entry.i16_next_step := FEHLER;
	(* Zylinder im Handbetrieb *)
	ELSIF gi16_betriebsart = HAND AND
		(st_visu.st_zyl.i16_nr_zyl_im_handbetrieb = zyl_wt_zentrierer_tisch.fb.st_config.i16_identnummer OR
		st_visu.st_zyl.i16_nr_zyl_im_handbetrieb = zyl_wt_stopper_tisch.fb.st_config.i16_identnummer)
		THEN
			fb_state_entry.i16_next_step := FEHLER;
	END_IF
END_IF

(* ============================Haupt-Schrittkette================================ *)
fb_state_entry(
	i16_next_step:= ,
	i16_pos:= 1,
	s_debugtext:= ,
	E=> ,
	X=> , 
	i16_step=> ,
	i16_last_step=> );

CASE fb_state_entry.i16_step OF
(*=======================================================*)
	INIT_OBJ:
		IF st_config.b_config_fertig THEN
			fb_state_entry.i16_next_step := INIT;
		END_IF

(*=======================================================*)
	INIT:
		IF fb_state_entry.E THEN
			fb_ton_wz.IN := FALSE;
			fb_ton_uez.IN := FALSE;
			fb_ton_quitt.IN := FALSE;
			st_ctrl_out.b_fehler := FALSE;
			st_ctrl_out.b_bereit := FALSE;
			st_ctrl_out.b_fertig := FALSE;
			st_ctrl_out.b_kontroller_start := FALSE;
			zyl_wt_zentrierer_tisch.st_ctrl.in.b_einfahren := FALSE;
			zyl_wt_zentrierer_tisch.st_ctrl.in.b_ausfahren := FALSE;
			zyl_wt_zentrierer_tisch.st_ctrl.in.b_luftlos := FALSE;
			zyl_wt_stopper_tisch.st_ctrl.in.b_einfahren := FALSE;
			zyl_wt_stopper_tisch.st_ctrl.in.b_ausfahren := FALSE;
			axis_z_achse.st_ctrl.in.b_start := FALSE;
			stueckzahlen.st_ctrl.in.b_gutteil_produziert := FALSE;
			sm_wt_hat_beladepos_nicht_verlassen := FALSE;
			sm_tagnummer_ungueltig := FALSE;
			sm_wt_hat_kein_tag := FALSE;
			sm_tagreader_nicht_fertig := FALSE;
			sm_keine_bandfreigabe := FALSE;
			bm_abfrage_wt_auf_beladepos := FALSE;
			bm_warte_auf_wt_an_stopper := FALSE;
			balluff_tag_reader.st_ctrl.in.b_start_lesen := FALSE;
			balluff_tag_reader.st_ctrl.in.b_start_schreiben := FALSE;

			bMerkerSchrittketteKommtVonInit := TRUE;
		END_IF

		(*-----------------------Weiterschaltbedingungen----------------------------*)
		IF st_ctrl_in.b_init THEN
			zyl_wt_zentrierer_tisch.st_ctrl.in.b_quittieren := FALSE;
			zyl_wt_stopper_tisch.st_ctrl.in.b_quittieren := FALSE;
			zyl_wt_zentrierer_tisch.st_ctrl.in.b_ausfahren := FALSE;
			fb_state_entry.i16_next_step := 20;
		END_IF

(*=======================================================*)
	20: (* Initialisierung: Stopper an Bestücktisch ausfahren und Zentrierer einfahren *)
		IF fb_state_entry.E THEN
			zyl_wt_stopper_tisch.st_ctrl.in.b_ausfahren := TRUE;
			zyl_wt_zentrierer_tisch.st_ctrl.in.b_einfahren := TRUE;
		END_IF

		(*-----------------------Weiterschaltbedingungen----------------------------*)
		IF zyl_wt_stopper_tisch.st_ctrl.out.b_ausgefahren AND zyl_wt_zentrierer_tisch.st_ctrl.out.b_eingefahren THEN
			zyl_wt_stopper_tisch.st_ctrl.in.b_ausfahren := FALSE;
			zyl_wt_zentrierer_tisch.st_ctrl.in.b_einfahren := FALSE;
			fb_state_entry.i16_next_step := BEREIT;
		END_IF

(*=======================================================*)
	BEREIT:	(* Warte auf Start von Kontroller *)
		IF fb_state_entry.E THEN
			st_ctrl_out.b_bereit := TRUE;
			st_ctrl_out.b_fertig := TRUE;
			stueckzahlen.st_ctrl.in.b_gutteil_produziert := FALSE;
		END_IF

	(*-----------------------Weiterschaltbedingungen----------------------------*)
		IF st_config.b_station_aktiv OR st_config.b_station_in_simulation THEN
			(* WT Transport aktiv oder in Simulation *)
			IF st_ctrl_in.b_start THEN
			(* WT Transport gestartet *)
				st_ctrl_out.b_fertig := FALSE;
				fb_ton_wz.IN := FALSE;
				st_ctrl_out.b_kontroller_start := TRUE;
				(* Abfrage, ob Schrittkette von Init kommt und ob WT auf Beladepos ist *)
				IF bMerkerSchrittketteKommtVonInit AND
					e_wt_auf_beladepos THEN
					fb_state_entry.i16_next_step := 170;	(* WT auslesen und prüfen, ob dieser schon bestückt wurde *)
				ELSE
					fb_state_entry.i16_next_step := 110;
				END_IF
			END_IF
		ELSE
			IF fb_r_trig_start.Q THEN
			(* Nur Z-Achse gestartet *)
				st_ctrl_out.b_fertig := FALSE;
				fb_ton_wz.IN := FALSE;
				fb_state_entry.i16_next_step := 500;
			END_IF
		END_IF

		IF fb_state_entry.X THEN
			bMerkerSchrittketteKommtVonInit := FALSE;
		END_IF

(*=======================================================*)
	110: (* WT-Abfrage auf Beladeposition *)
		IF fb_state_entry.E THEN
			bm_abfrage_wt_auf_beladepos := TRUE;
		END_IF

		(*-----------------------Weiterschaltbedingungen----------------------------*)
		IF e_wt_auf_beladepos THEN
			(* Ein WT ist anwesend zum rausschicken *)
			IF NOT ST_WT_Transport_Abgabe.e_wt_auf_abgabepos THEN
				(* Erst wenn kein Stau vorhanden ist, dann wird der WT weiter gelassen *)
				st_ctrl_out.b_kontroller_start := FALSE;
				bm_abfrage_wt_auf_beladepos := FALSE;
				fb_state_entry.i16_next_step := 120;
			END_IF
		ELSE	(* Kein WT da, deshalb einen holen *)
			st_ctrl_out.b_kontroller_start := FALSE;
			bm_abfrage_wt_auf_beladepos := FALSE;
			fb_state_entry.i16_next_step := 140;
		END_IF

(*=======================================================*)
	120: (* WT-Zentrierer und Stopper einfahren *)
		IF fb_state_entry.E THEN
			zyl_wt_stopper_tisch.st_ctrl.in.b_einfahren := TRUE;
			zyl_wt_zentrierer_tisch.st_ctrl.in.b_einfahren := TRUE;
			fb_Zentrierer_einfahren(b_start:= TRUE, t_zeit=> );
		END_IF
		IF 	zyl_wt_zentrierer_tisch.st_ctrl.out.b_eingefahren THEN
			fb_Zentrierer_einfahren(b_start:= FALSE, t_zeit=>t_Zentrierer_einfahren );
		END_IF

		(*-----------------------Weiterschaltbedingungen----------------------------*)
		IF zyl_wt_stopper_tisch.st_ctrl.out.b_eingefahren AND zyl_wt_zentrierer_tisch.st_ctrl.out.b_eingefahren THEN
			zyl_wt_stopper_tisch.st_ctrl.in.b_einfahren := FALSE;
			zyl_wt_zentrierer_tisch.st_ctrl.in.b_einfahren := FALSE;
			fb_state_entry.i16_next_step := 130;
		END_IF

(*=======================================================*)
	130: (* Und auf Pufferstrecke angekommen ist *)
		IF fb_state_entry.E THEN
			fb_ton_uez.PT := t#5s;
 			fb_ton_uez.IN := TRUE;
		END_IF

		(*-----------------------Weiterschaltbedingungen----------------------------*)
		IF fb_r_trig_beladepos_verlassen.Q THEN
			fb_ton_uez.IN := FALSE;
			fb_state_entry.i16_next_step := 140;
		ELSIF fb_ton_uez.Q THEN
			sm_wt_hat_beladepos_nicht_verlassen := TRUE;
			fb_state_entry.i16_next_step := FEHLER;
		END_IF

(*=======================================================*)
	140: (* Stopper ausfahren und  WT-Zentrierer einfahren *)
		IF fb_state_entry.E THEN
			zyl_wt_stopper_tisch.st_ctrl.in.b_ausfahren := TRUE;
			zyl_wt_zentrierer_tisch.st_ctrl.in.b_einfahren := TRUE;
		END_IF

		(*-----------------------Weiterschaltbedingungen----------------------------*)
		IF 	zyl_wt_stopper_tisch.st_ctrl.out.b_ausgefahren AND
			zyl_wt_zentrierer_tisch.st_ctrl.out.b_eingefahren
			THEN
				zyl_wt_stopper_tisch.st_ctrl.in.b_ausfahren := FALSE;
				zyl_wt_zentrierer_tisch.st_ctrl.in.b_einfahren := FALSE;
				st_ctrl_out.b_kontroller_start := TRUE;
				fb_state_entry.i16_next_step := 150;
		END_IF

(*=======================================================*)
	150: (* Warte auf Flanke "angekommen an Tisch-Stopper" *)
		IF fb_state_entry.E THEN
			bm_warte_auf_wt_an_stopper := TRUE;
		END_IF

		(*-----------------------Weiterschaltbedingungen----------------------------*)
		IF  fb_r_trig_beladepos.Q THEN
			st_ctrl_out.b_kontroller_start := FALSE;
			fb_state_entry.i16_next_step := 160;
		END_IF

(*=======================================================*)
	160: (* WT sicher angekommen an Tisch-Stopper *)

		(*-----------------------Weiterschaltbedingungen----------------------------*)
		IF  fb_ton_wt_auf_beladepos.Q THEN
			bm_warte_auf_wt_an_stopper := FALSE;
			fb_state_entry.i16_next_step := 170;
		END_IF

(*=======================================================*)
	170: (* WT-Zentrierer ausfahren *)
		IF fb_state_entry.E THEN
			zyl_wt_zentrierer_tisch.st_ctrl.in.b_ausfahren := TRUE;
			fb_Zentrierer_ausfahren(b_start:= TRUE, t_zeit=> );
		END_IF

		(*-----------------------Weiterschaltbedingungen----------------------------*)
		IF zyl_wt_zentrierer_tisch.st_ctrl.out.b_ausgefahren AND
			NOT ST_TippTasten.b_einfaedeln_aktiv AND
			NOT ST_Virtuelle_Masterachse.b_merker_bandende_links  AND
 			NOT ST_Virtuelle_Masterachse.b_merker_bandende_rechts THEN
			fb_Zentrierer_ausfahren(b_start:= FALSE, t_zeit=> t_Zentrierer_ausfahren);
			zyl_wt_zentrierer_tisch.st_ctrl.in.b_ausfahren := FALSE;
			IF st_config.b_station_in_simulation THEN
				(* WT-Transport ist in Simulation und deshalb wird der WT ohne zu Bestücken weiter gefahren *)
				fb_state_entry.i16_next_step := BEREIT;
			ELSE
				fb_state_entry.i16_next_step := 180;
			END_IF
		END_IF

(*=======================================================*)
	180: (* WT-Tag mit RFID-Lesegerät abfragen *)
		IF fb_state_entry.E THEN
			fb_ton_wz.PT := t#100ms;
			fb_ton_wz.IN := TRUE;
		END_IF

		(*-----------------------Weiterschaltbedingungen----------------------------*)
		IF fb_ton_wz.Q THEN
			IF e_wt_im_aktionsfeld THEN
				(* Tag auslesen *)
				fb_ton_wz.IN := FALSE;
				fb_state_entry.i16_next_step := 230;
			ELSE
				(* Kein Tag auf WT *)
				sm_wt_hat_kein_tag := TRUE;
				fb_state_entry.i16_next_step := FEHLER;
			END_IF
		END_IF

(*=======================================================*)
	230: (* Z-Achse und anschliessend Bestückachse wird gestartet *)
		IF fb_state_entry.E THEN
			axis_z_achse.st_ctrl.in.b_start := TRUE;
			(*Zeitmessung Trägerwechsel stoppen und ausgeben*)
			fb_WT_WechselZeit(b_start:=FALSE , t_zeit=>t_WT_WechselZeit );
		END_IF

		(*-----------------------Weiterschaltbedingungen----------------------------*)
		(*IF axis_bestueckachse.st_ctrl.in.b_start THEN*)
		IF	axis_virt_master.st_ctrl.in.b_start THEN
			fb_state_entry.i16_next_step := 240;
		END_IF

		(*WT abgeben bei NIO*)
		IF axis_z_achse.st_ctrl.out.b_fertig AND NOT fb_state_entry.E THEN
			axis_z_achse.st_ctrl.in.b_start := FALSE;
			st_ctrl_out.b_kontroller_start := FALSE;
			fb_state_entry.i16_next_step := BEREIT;
		END_IF


(*=======================================================*)
	240: (* WT-Zentrierzylinder luftlos machen *)
		IF fb_state_entry.E THEN
			zyl_wt_zentrierer_tisch.st_ctrl.in.b_luftlos := TRUE;
		END_IF

		(*-----------------------Weiterschaltbedingungen----------------------------*)
		IF zyl_wt_zentrierer_tisch.st_ctrl.out.b_ohne_luft THEN
			(* Luftlos-Kommando bleibt TRUE, und für die Überwachung brauchen wir noch das Ausfahr-Kommando *)
			zyl_wt_zentrierer_tisch.st_ctrl.in.b_ausfahren := TRUE;
			fb_state_entry.i16_next_step := 250;
		END_IF

(*=======================================================*)
	250: (* Bestückachse ist fertig *)

		(*-----------------------Weiterschaltbedingungen----------------------------*)
		IF axis_virt_master.st_ctrl.out.b_fertig = TRUE THEN
			zyl_wt_zentrierer_tisch.st_ctrl.in.b_luftlos := FALSE;
			fb_state_entry.i16_next_step := 260;
		END_IF

(*=======================================================*)
	260: (* WT-Zentrierer ausfahren *)
		IF fb_state_entry.E THEN
			zyl_wt_zentrierer_tisch.st_ctrl.in.b_ausfahren := TRUE;
		END_IF

		(*-----------------------Weiterschaltbedingungen----------------------------*)
		IF zyl_wt_zentrierer_tisch.st_ctrl.out.b_ausgefahren THEN
			zyl_wt_zentrierer_tisch.st_ctrl.in.b_ausfahren := FALSE;
			fb_state_entry.i16_next_step := 270;
		END_IF

(*=======================================================*)
	270: (* Z-Achse ist fertig *)

		(*-----------------------Weiterschaltbedingungen----------------------------*)
		IF axis_z_achse.st_ctrl.out.b_fertig AND NOT fb_state_entry.E THEN
			(*Zeitmessung Trägerwechsel starten*)
			fb_WT_WechselZeit(b_start:=TRUE , t_zeit=> );
			(*Zeitmessung zusammenfassen*)
			t_bestueckzeit:=ST_Z_Achse.t_Bestueckung;
			t_traegerwechselzeit:=t_WT_WechselZeit + ST_Z_Achse.t_Z_Achse_einfahren + ST_Z_Achse.t_Z_Achse_ausfahren;
			t_komplett_zyklus:= t_traegerwechselzeit + t_bestueckzeit;

			axis_z_achse.st_ctrl.in.b_start := FALSE;
			stueckzahlen.st_ctrl.in.b_gutteil_produziert := TRUE;
			fb_state_entry.i16_next_step := BEREIT;
		END_IF

		IF fb_state_entry.X THEN
			gst_datensatz.st_md.produzierte_Stecker := gst_datensatz.st_md.produzierte_Stecker + 1;
		END_IF

(*=======================================================*)
	500: (* Warte bis angekommen an Stopper *)

		(*-----------------------Weiterschaltbedingungen----------------------------*)
		IF fb_ton_wt_auf_beladepos.Q THEN
			fb_state_entry.i16_next_step := 510;
		END_IF

(*=======================================================*)
	510: (* WT-Zentrierer auf Bestücktisch ausfahren *)
		IF fb_state_entry.E THEN
			zyl_wt_zentrierer_tisch.st_ctrl.in.b_ausfahren := TRUE;
		END_IF

		(*-----------------------Weiterschaltbedingungen----------------------------*)
		IF zyl_wt_zentrierer_tisch.st_ctrl.out.b_ausgefahren  THEN
			zyl_wt_zentrierer_tisch.st_ctrl.in.b_ausfahren := FALSE;
			axis_z_achse.st_ctrl.in.b_start := TRUE;
			fb_state_entry.i16_next_step := 520;
		END_IF

(*=======================================================*)
	520: (* Bestückachse wird gestartet *)

		(*-----------------------Weiterschaltbedingungen----------------------------*)
		IF axis_virt_master.st_ctrl.in.b_start THEN
			fb_state_entry.i16_next_step := 530;
		END_IF

(*=======================================================*)
	530: (* WT-Zentrierzylinder luftlos machen *)
		IF fb_state_entry.E THEN
			zyl_wt_zentrierer_tisch.st_ctrl.in.b_luftlos := TRUE;
		END_IF

		(*-----------------------Weiterschaltbedingungen----------------------------*)
		IF zyl_wt_zentrierer_tisch.st_ctrl.out.b_ohne_luft THEN
			(* Luftlos-Kommando bleibt TRUE, und für die Überwachung brauchen wir noch das Ausfahr-Kommando *)
			zyl_wt_zentrierer_tisch.st_ctrl.in.b_ausfahren := TRUE;
			fb_state_entry.i16_next_step := 540;
		END_IF

(*=======================================================*)
	540: (* Bestückablauf ist fertig *)

		(*-----------------------Weiterschaltbedingungen----------------------------*)
		IF axis_virt_master.st_ctrl.out.b_fertig THEN
			zyl_wt_zentrierer_tisch.st_ctrl.in.b_luftlos := FALSE;
			fb_state_entry.i16_next_step := 550;
		END_IF

(*=======================================================*)
	550: (* WT-Zentrierer ausfahren *)
		IF fb_state_entry.E THEN
			zyl_wt_zentrierer_tisch.st_ctrl.in.b_ausfahren := TRUE;
		END_IF

		(*-----------------------Weiterschaltbedingungen----------------------------*)
		IF zyl_wt_zentrierer_tisch.st_ctrl.out.b_ausgefahren THEN
			zyl_wt_zentrierer_tisch.st_ctrl.in.b_ausfahren := FALSE;
			fb_state_entry.i16_next_step := 560;
		END_IF

(*=======================================================*)
	560:	(* Warte auf Z-Achse komplett fertig *)

		(*-----------------------Weiterschaltbedingungen----------------------------*)
		IF axis_z_achse.st_ctrl.out.b_fertig AND NOT fb_state_entry.E THEN
			axis_z_achse.st_ctrl.in.b_start := FALSE;
			stueckzahlen.st_ctrl.in.b_gutteil_produziert := TRUE;
			IF NOT b_Dauertest_Achsen THEN
				fb_state_entry.i16_next_step := BEREIT;
			ELSE
				(* zum Testen der Achsen nach Tausch, Bestückbild "Becherspucken", WKZ ausgebaut, Vorschubkontrolle abeschaltet,
				Bit muss von Programmierer geforct werden, zum Beenden Schlüsselschalter auf HAND und Zelle neu starten *)
				fb_state_entry.i16_next_step := 500;	(* Dauertest *)
			END_IF
		END_IF

		IF fb_state_entry.X AND NOT b_Dauertest_Achsen THEN
			gst_datensatz.st_md.produzierte_Stecker := gst_datensatz.st_md.produzierte_Stecker + 1;
		END_IF

(*=======================================================*)
	FEHLER:
		IF fb_state_entry.E THEN
			st_ctrl_out.b_fehler := TRUE;
			fb_ton_quitt.IN := FALSE;
			zyl_wt_zentrierer_tisch.st_ctrl.in.b_quittieren := FALSE;
			zyl_wt_stopper_tisch.st_ctrl.in.b_quittieren := FALSE;

			(*ST_Markiere_WT_NIO();*)
		END_IF

		(*-----------------------Weiterschaltbedingungen----------------------------*)
		IF st_ctrl_in.b_quitt AND NOT fb_state_entry.E THEN
			st_ctrl_out.b_fehler := FALSE;
			zyl_wt_zentrierer_tisch.st_ctrl.in.b_quittieren := TRUE;
			zyl_wt_stopper_tisch.st_ctrl.in.b_quittieren := TRUE;
			fb_ton_quitt.IN := TRUE;
		END_IF

		IF fb_ton_quitt.Q THEN
			fb_ton_quitt.IN := FALSE;
			fb_state_entry.i16_next_step := INIT;
		END_IF

(*=======================================================*)
	STOP:
		IF fb_state_entry.E THEN
			fb_ton_quitt.IN := FALSE;
			st_ctrl_out.b_kontroller_start := FALSE;
			zyl_wt_zentrierer_tisch.st_ctrl.in.b_quittieren := FALSE;
			zyl_wt_stopper_tisch.st_ctrl.in.b_quittieren := FALSE;
			(*ST_Markiere_WT_NIO();*)
		END_IF

		(*-----------------------Weiterschaltbedingungen----------------------------*)
		IF st_ctrl_in.b_quitt AND NOT fb_state_entry.E THEN
			fb_ton_quitt.IN := TRUE;
			zyl_wt_zentrierer_tisch.st_ctrl.in.b_quittieren := TRUE;
			zyl_wt_stopper_tisch.st_ctrl.in.b_quittieren := TRUE;
		END_IF

		IF fb_ton_quitt.Q THEN
			fb_ton_quitt.IN := FALSE;
			fb_state_entry.i16_next_step := INIT;
		END_IF
END_CASE

fb_state_entry(
	i16_next_step:= ,
	i16_pos:= 2,
	s_debugtext:= ,
	E=> ,
	X=> ,
	i16_step=> ,
	i16_last_step=> );

fb_ton_abfrage_wt_auf_beladepos (IN:=bm_abfrage_wt_auf_beladepos,PT:=t#30s);
fb_ton_warte_auf_wt_an_stopper (IN:=bm_warte_auf_wt_an_stopper,PT:=t#30s);

IF st_config.b_config_fertig THEN
	(* Fehlermeldungen ab dem Startindex in das globale Störmeldungsarray schreiben *)
	garr_stoermeldungen[st_config.i16_meld_startindex + 0] := sm_wt_hat_beladepos_nicht_verlassen;
	garr_stoermeldungen[st_config.i16_meld_startindex + 1] := sm_tagnummer_ungueltig;
	garr_stoermeldungen[st_config.i16_meld_startindex + 2] := sm_wt_hat_kein_tag;
	garr_stoermeldungen[st_config.i16_meld_startindex + 3] := FALSE;
	garr_stoermeldungen[st_config.i16_meld_startindex + 4] := sm_tagreader_nicht_fertig;
	garr_stoermeldungen[st_config.i16_meld_startindex + 5] := sm_keine_bandfreigabe;
	garr_stoermeldungen[st_config.i16_meld_startindex + 6] := FALSE;
	garr_stoermeldungen[st_config.i16_meld_startindex + 7] := FALSE;
	garr_stoermeldungen[st_config.i16_meld_startindex + 8] := FALSE;
	garr_stoermeldungen[st_config.i16_meld_startindex + 9] := FALSE;
	garr_stoermeldungen[st_config.i16_meld_startindex + 10] := FALSE;
	garr_stoermeldungen[st_config.i16_meld_startindex + 11] := FALSE;
	garr_stoermeldungen[st_config.i16_meld_startindex + 12] := FALSE;
	garr_stoermeldungen[st_config.i16_meld_startindex + 13] := FALSE;
	garr_stoermeldungen[st_config.i16_meld_startindex + 14] := FALSE;
	garr_stoermeldungen[st_config.i16_meld_startindex + 15] := FALSE;
	garr_stoermeldungen[st_config.i16_meld_startindex + 16] := FALSE;
	garr_stoermeldungen[st_config.i16_meld_startindex + 17] := FALSE;
	garr_stoermeldungen[st_config.i16_meld_startindex + 18] := FALSE;
	garr_stoermeldungen[st_config.i16_meld_startindex + 19] := FALSE;
	
	garr_betriebsmeldungen[st_config.i16_meld_startindex + 0] := fb_ton_abfrage_wt_auf_beladepos.Q;
	garr_betriebsmeldungen[st_config.i16_meld_startindex + 1] := fb_ton_warte_auf_wt_an_stopper.Q;
	garr_betriebsmeldungen[st_config.i16_meld_startindex + 2] := FALSE;
	garr_betriebsmeldungen[st_config.i16_meld_startindex + 3] := FALSE;
	garr_betriebsmeldungen[st_config.i16_meld_startindex + 4] := FALSE;
	garr_betriebsmeldungen[st_config.i16_meld_startindex + 5] := FALSE;
	garr_betriebsmeldungen[st_config.i16_meld_startindex + 6] := FALSE;
	garr_betriebsmeldungen[st_config.i16_meld_startindex + 7] := FALSE;
	garr_betriebsmeldungen[st_config.i16_meld_startindex + 8] := FALSE;
	garr_betriebsmeldungen[st_config.i16_meld_startindex + 9] := FALSE;
	garr_betriebsmeldungen[st_config.i16_meld_startindex + 10] := FALSE;
	garr_betriebsmeldungen[st_config.i16_meld_startindex + 11] := FALSE;
	garr_betriebsmeldungen[st_config.i16_meld_startindex + 12] := FALSE;
	garr_betriebsmeldungen[st_config.i16_meld_startindex + 13] := FALSE;
	garr_betriebsmeldungen[st_config.i16_meld_startindex + 14] := FALSE;
	garr_betriebsmeldungen[st_config.i16_meld_startindex + 15] := FALSE;
	garr_betriebsmeldungen[st_config.i16_meld_startindex + 16] := FALSE;
	garr_betriebsmeldungen[st_config.i16_meld_startindex + 17] := FALSE;
	garr_betriebsmeldungen[st_config.i16_meld_startindex + 18] := FALSE;
	garr_betriebsmeldungen[st_config.i16_meld_startindex + 19] := FALSE;
END_IF
END_PROGRAM

(* POU Gemeinsamkeiten17xx/WT Transport/ST_WT_Transport_Abgabe, ST *)
PROGRAM ST_WT_Transport_Abgabe
VAR_INPUT
	st_config								: struct_config;
	st_ctrl_in								: struct_ctrl_in;
	e_station_nachher_in_erlaubnis			: BOOL := FALSE;
	e_station_nachher_in_angekommen		: BOOL := FALSE;
END_VAR
VAR_IN_OUT
	st_visu								: struct_visu;
END_VAR
VAR_OUTPUT
	st_ctrl_out							: struct_ctrl_out;
	a_station_nachher_out_anforderung		: BOOL := FALSE;
	a_station_nachher_out_abgegeben		: BOOL := FALSE;
END_VAR
VAR
	fb_ton_uez							: TON;
	fb_ton_wz							: TON;
	fb_ton_quitt							: TON;
	fb_ton_wt_auf_abgabepos				: TON;
	fb_tof_wt_auf_abgabepos				: TOF;
	fb_WT_WechselZeit					: ST_Taktzeit;
	t_traegerwechselzeit					: TIME := t#0ms;
	t_traegerwechselzeit_help				: TIME := t#0ms;
	fb_f_trig_abgabepos					: F_TRIG;
	fb_r_trig_start							: R_TRIG;
	fb_r_trig_pm_time						: R_TRIG;
	fb_state_entry							: ST_StateEntry;
	i16_state_msg						: INT;
	sm_wt_hat_abgabepos_nicht_verlassen	: BOOL := FALSE;
	sm_wt_hat_abgabepos_ueberfahren		: BOOL := FALSE;
	bm_setze_anforderung					: BOOL := FALSE;
	bm_abfrage_wt_an_stopper				: BOOL := FALSE;
	pm_traegerwechselzeit					: BOOL := FALSE;
	e_wt_auf_abgabepos					AT %I* : BOOL;
	e_wt_abgabepos_verlassen			AT %I* : BOOL;
END_VAR
(* Zeiten *)
fb_ton_uez(IN:= , PT:= , Q=>  , ET=> );
fb_ton_wz(IN:= , PT:= , Q=> , ET=> );
fb_ton_quitt(IN:= , PT:= t#100ms, Q=> , ET=> );
fb_WT_WechselZeit(b_start:= , t_zeit=> );

fb_ton_wt_auf_abgabepos(IN:= e_wt_auf_abgabepos, PT:= t#500ms, Q=> , ET=> );
fb_tof_wt_auf_abgabepos(IN:=e_wt_auf_abgabepos , PT:= t#200ms, Q=> , ET=> );

(* Flanken *)
fb_f_trig_abgabepos(CLK:= e_wt_auf_abgabepos, Q=> );
fb_r_trig_start(CLK:= st_ctrl_in.b_start, Q=> );


(*Meldung für Trägerwechselzeit zu groß nur ausgeben, wenn Hublift nicht aktiv ist*)
IF NOT gst_Datensatz.st_md.b_hublift_rechts_aktiv THEN
	fb_r_trig_pm_time(CLK:= pm_traegerwechselzeit, Q=> );
END_IF

IF fb_r_trig_pm_time.Q  THEN
	t_traegerwechselzeit_help := t_traegerwechselzeit;
	i16_state_msg := 1;
END_IF

(*Produktionsmeldung für Übergabe zu lange*)
CASE i16_state_msg OF
	1: (*Warten bis keine ander Produktions Meldung ansteht *)
		IF	TestAndSet(ST_Message_Produktion.LockFlag) THEN
			ST_Message_Produktion.ClearMessageLines();
			i16_state_msg := 2;
		END_IF

	2:  (*Produktions Meldung*)
		Visu.MeldungProduktion.Color_R := 255;
		Visu.MeldungProduktion.Color_G := 255;
		Visu.MeldungProduktion.Color_B := 0;
		IF visu.s_akt_sprache = 'de' THEN
			Visu.MeldungProduktion.Name:=CONCAT('WT Wechsel in die nächste Zelle hat zu lange gedautert.',TIME_TO_STRING(t_traegerwechselzeit_help));
		ELSIF visu.s_akt_sprache = 'en' THEN
			Visu.MeldungProduktion.Name:=CONCAT('carrier exchange into station exceeded time limit.',TIME_TO_STRING(t_traegerwechselzeit_help));
		ELSIF visu.s_akt_sprache = 'cz' THEN
			Visu.MeldungProduktion.Name:=CONCAT('Prejezd paletky do dalsi cely trval prilis dlouho.',TIME_TO_STRING(t_traegerwechselzeit_help));
		END_IF
		Visu.MeldungProduktion.ShowMessage := TRUE;
		Visu.MeldungProduktion.Button1.sichtbar:=TRUE;	(*OK*)
		Visu.MeldungProduktion.Button1.Text:='Ok';
		i16_state_msg := 3;

	3:  (*Warte auf OK*)
		IF Visu.MeldungProduktion.Button1.tasten THEN
			i16_state_msg:=0;
		END_IF
END_CASE

(* Toplevel *)
IF fb_state_entry.i16_next_step > INIT AND fb_state_entry.i16_next_step < FEHLER THEN
	IF fb_state_entry.i16_next_step < STOP THEN
		IF st_ctrl_in.b_stop THEN
			fb_state_entry.i16_next_step := STOP;
		END_IF
	END_IF

	(* Allgemeine Fehler *)
	IF zyl_wt_stopper_auslauf.st_ctrl.out.b_fehler THEN
		fb_state_entry.i16_next_step := FEHLER;

	(* Zylinder im Handbetrieb *)
	ELSIF gi16_betriebsart = HAND AND
		(st_visu.st_zyl.i16_nr_zyl_im_handbetrieb = zyl_wt_stopper_auslauf.fb.st_config.i16_identnummer )
		THEN
			fb_state_entry.i16_next_step := FEHLER;
	END_IF
END_IF


(* ==================================Schrittkette================================ *)
fb_state_entry(
	i16_next_step:= ,
	i16_pos:= 1,
	s_debugtext:= ,
	E=> ,
	X=> ,
	i16_step=> ,
	i16_last_step=> );

CASE fb_state_entry.i16_step OF
(*=======================================================*)
	INIT_OBJ:
		IF st_config.b_config_fertig THEN
			fb_state_entry.i16_next_step := INIT;
		END_IF

(*=======================================================*)
	INIT:
		IF fb_state_entry.E THEN
			fb_ton_wz.IN := FALSE;
			fb_ton_uez.IN := FALSE;
			fb_ton_quitt.IN := FALSE;
			st_ctrl_out.b_fehler := FALSE;
			st_ctrl_out.b_bereit := FALSE;
			st_ctrl_out.b_fertig := FALSE;
			st_ctrl_out.b_kontroller_start := FALSE;
			zyl_wt_stopper_auslauf.st_ctrl.in.b_einfahren := FALSE;
			zyl_wt_stopper_auslauf.st_ctrl.in.b_ausfahren := FALSE;
			sm_wt_hat_abgabepos_nicht_verlassen := FALSE;
			sm_wt_hat_abgabepos_ueberfahren := FALSE;
			bm_setze_anforderung := FALSE;
			bm_abfrage_wt_an_stopper := FALSE;
			a_station_nachher_out_anforderung := FALSE;
			a_station_nachher_out_abgegeben := FALSE;
		END_IF

		(*-----------------------Weiterschaltbedingungen----------------------------*)
		IF st_ctrl_in.b_init THEN
			zyl_wt_stopper_auslauf.st_ctrl.in.b_quittieren := FALSE;
			fb_state_entry.i16_next_step := 20;
		END_IF

(*=======================================================*)
	20: (* Initialisierung: Auslaufstopper ausfahren *)
		IF fb_state_entry.E THEN
			zyl_wt_stopper_auslauf.st_ctrl.in.b_ausfahren := TRUE;
		END_IF

		(*-----------------------Weiterschaltbedingungen----------------------------*)
		IF zyl_wt_stopper_auslauf.st_ctrl.out.b_ausgefahren THEN
			zyl_wt_stopper_auslauf.st_ctrl.in.b_ausfahren := FALSE;
			fb_state_entry.i16_next_step := BEREIT;
		END_IF

(*=======================================================*)
	BEREIT:	(* Warte auf Startfreigabe von Kontroller *)
		IF fb_state_entry.E THEN
			st_ctrl_out.b_bereit := TRUE;
			st_ctrl_out.b_fertig := TRUE;
		END_IF

	(*-----------------------Weiterschaltbedingungen----------------------------*)
		IF st_config.b_station_aktiv OR st_config.b_station_in_simulation THEN
			(* WT Transport aktiv oder in Simulation *)
			IF st_ctrl_in.b_start THEN
				fb_state_entry.i16_next_step := 110;
			END_IF
		ELSE
			(* WT Transport nicht aktiv und nicht in Simulation -> tue nichts  *)
 			;
		END_IF

(*=======================================================*)
	110: (* Statische WT-Abfrage auf Abgabeposition *)
		IF fb_state_entry.E THEN
			st_ctrl_out.b_kontroller_start := TRUE;
			bm_abfrage_wt_an_stopper := TRUE;
		END_IF

		(*-----------------------Weiterschaltbedingungen----------------------------*)
		IF e_wt_auf_abgabepos THEN
			st_ctrl_out.b_kontroller_start := FALSE;
			bm_abfrage_wt_an_stopper := FALSE;
			fb_state_entry.i16_next_step := 120;
		END_IF

(*=======================================================*)
	120:  (* Setze Anforderung an folgende Station *)
		IF fb_state_entry.E THEN
			a_station_nachher_out_anforderung := TRUE;
			bm_setze_anforderung := TRUE;
		END_IF

		(*-----------------------Weiterschaltbedingungen----------------------------*)
		IF e_station_nachher_in_erlaubnis  AND NOT fb_state_entry.E THEN
			bm_setze_anforderung := FALSE;
			fb_state_entry.i16_next_step := 130;
		ELSIF e_wt_abgabepos_verlassen THEN
			(* Abgabeposition wurde unerlaubterweise überfahren *)
			sm_wt_hat_abgabepos_ueberfahren := TRUE;
			fb_state_entry.i16_next_step := FEHLER;
		END_IF

(*=======================================================*)
	130: (* WT-Stopper einfahren *)
		IF fb_state_entry.E THEN
			st_ctrl_out.b_kontroller_start := TRUE;
			zyl_wt_stopper_auslauf.st_ctrl.in.b_einfahren := TRUE;
			fb_WT_WechselZeit(b_start:=TRUE , t_zeit=> );
			pm_traegerwechselzeit := FALSE;
		END_IF

		(*-----------------------Weiterschaltbedingungen----------------------------*)
		IF zyl_wt_stopper_auslauf.st_ctrl.out.b_eingefahren OR e_wt_abgabepos_verlassen (* wegen möglichen Problemen beim schnellen Förderband*)THEN
			zyl_wt_stopper_auslauf.st_ctrl.in.b_einfahren := FALSE;
			st_ctrl_out.b_kontroller_start := FALSE;
			fb_state_entry.i16_next_step := 140;
		END_IF

(*=======================================================*)
	140: (* Warte bis WT an "verlassen" Sensor *)
		IF fb_state_entry.E THEN
			fb_ton_uez.PT := t#300ms;
 			fb_ton_uez.IN := TRUE;
			st_ctrl_out.b_kontroller_start := TRUE;
		END_IF

		(*-----------------------Weiterschaltbedingungen----------------------------*)
		IF ST_Hublift_rechts.st_config.b_station_aktiv THEN
			st_ctrl_out.b_kontroller_start := TRUE;
			IF	 e_wt_abgabepos_verlassen THEN
				(* Bei Hublift kann der WT den Sensor nicht erreichen, deshalb gleich Meldung an nachfolgende Station *)
 				fb_ton_uez.IN := FALSE;
				fb_state_entry.i16_next_step := 150;
			ELSIF fb_ton_uez.Q THEN
				sm_wt_hat_abgabepos_nicht_verlassen := TRUE;
				fb_state_entry.i16_next_step := FEHLER;
			END_IF
		ELSE
			st_ctrl_out.b_kontroller_start := FALSE;
			IF e_wt_abgabepos_verlassen THEN
	 			fb_ton_uez.IN := FALSE;
				a_station_nachher_out_abgegeben := TRUE;
				fb_state_entry.i16_next_step := 150;
			ELSIF fb_ton_uez.Q THEN
				sm_wt_hat_abgabepos_nicht_verlassen := TRUE;
				fb_state_entry.i16_next_step := FEHLER;
			END_IF
		END_IF

(*=======================================================*)
	150: (* Auslaufstopper ausfahren *)
		IF fb_state_entry.E THEN
			zyl_wt_stopper_auslauf.st_ctrl.in.b_ausfahren := TRUE;
		END_IF

		(*-----------------------Weiterschaltbedingungen----------------------------*)
		IF zyl_wt_stopper_auslauf.st_ctrl.out.b_ausgefahren THEN
			zyl_wt_stopper_auslauf.st_ctrl.in.b_ausfahren := FALSE;
			fb_state_entry.i16_next_step := 160;
		END_IF

(*=======================================================*)
	160: (* Warte bis die folgende Station "angekommen" meldet *)
		IF fb_state_entry.E THEN
			a_station_nachher_out_abgegeben := FALSE;
			st_ctrl_out.b_kontroller_start := TRUE;
		END_IF

		(*-----------------------Weiterschaltbedingungen----------------------------*)
		IF e_station_nachher_in_angekommen THEN
			fb_WT_WechselZeit(b_start:=FALSE , t_zeit=>t_traegerwechselzeit );
			a_station_nachher_out_anforderung := FALSE;
			st_ctrl_out.b_kontroller_start := FALSE;
			pm_traegerwechselzeit := t_traegerwechselzeit > gst_datensatz.st_md.t_max_traegerwechselzeit AND gst_datensatz.st_md.t_max_traegerwechselzeit <> INT_TO_TIME(0);
			fb_state_entry.i16_next_step := BEREIT;
		END_IF

(*=======================================================*)
	FEHLER:
		IF fb_state_entry.E THEN
			st_ctrl_out.b_fehler := TRUE;
			fb_ton_quitt.IN := FALSE;
			zyl_wt_stopper_auslauf.st_ctrl.in.b_quittieren := FALSE;
			a_station_nachher_out_anforderung := FALSE;
			a_station_nachher_out_abgegeben := FALSE;
		END_IF

		(*-----------------------Weiterschaltbedingungen----------------------------*)
		IF st_ctrl_in.b_quitt AND NOT fb_state_entry.E THEN
			st_ctrl_out.b_fehler := FALSE;
			zyl_wt_stopper_auslauf.st_ctrl.in.b_quittieren := TRUE;
			fb_ton_quitt.IN := TRUE;
		END_IF

		IF fb_ton_quitt.Q THEN
			fb_ton_quitt.IN := FALSE;
			fb_state_entry.i16_next_step := INIT;
		END_IF

(*=======================================================*)
	STOP:
		IF fb_state_entry.E THEN
			fb_ton_quitt.IN := FALSE;
			st_ctrl_out.b_kontroller_start := FALSE;
			zyl_wt_stopper_auslauf.st_ctrl.in.b_quittieren := FALSE;
			a_station_nachher_out_anforderung := FALSE;
			a_station_nachher_out_abgegeben := FALSE;
		END_IF

		(*-----------------------Weiterschaltbedingungen----------------------------*)
		IF st_ctrl_in.b_quitt AND NOT fb_state_entry.E THEN
			fb_ton_quitt.IN := TRUE;
			zyl_wt_stopper_auslauf.st_ctrl.in.b_quittieren := TRUE;
		END_IF

		IF fb_ton_quitt.Q THEN
			fb_ton_quitt.IN := FALSE;
			fb_state_entry.i16_next_step := INIT;
		END_IF
END_CASE

fb_state_entry(
	i16_next_step:= ,
	i16_pos:= 2,
	s_debugtext:= ,
	E=> ,
	X=> ,
	i16_step=> ,
	i16_last_step=> );

IF st_config.b_config_fertig THEN
	(* Fehlermeldungen ab dem Startindex in das globale Störmeldungsarray schreiben *)
	garr_stoermeldungen[st_config.i16_meld_startindex + 0] := sm_wt_hat_abgabepos_nicht_verlassen;
	garr_stoermeldungen[st_config.i16_meld_startindex + 1] := sm_wt_hat_abgabepos_ueberfahren;
	garr_stoermeldungen[st_config.i16_meld_startindex + 2] := FALSE;
	garr_stoermeldungen[st_config.i16_meld_startindex + 3] := FALSE;
	garr_stoermeldungen[st_config.i16_meld_startindex + 4] := FALSE;
	garr_stoermeldungen[st_config.i16_meld_startindex + 5] := FALSE;
	garr_stoermeldungen[st_config.i16_meld_startindex + 6] := FALSE;
	garr_stoermeldungen[st_config.i16_meld_startindex + 7] := FALSE;
	garr_stoermeldungen[st_config.i16_meld_startindex + 8] := FALSE;
	garr_stoermeldungen[st_config.i16_meld_startindex + 9] := FALSE;
	garr_stoermeldungen[st_config.i16_meld_startindex + 10] := FALSE;
	garr_stoermeldungen[st_config.i16_meld_startindex + 11] := FALSE;
	garr_stoermeldungen[st_config.i16_meld_startindex + 12] := FALSE;
	garr_stoermeldungen[st_config.i16_meld_startindex + 13] := FALSE;
	garr_stoermeldungen[st_config.i16_meld_startindex + 14] := FALSE;
	garr_stoermeldungen[st_config.i16_meld_startindex + 15] := FALSE;
	garr_stoermeldungen[st_config.i16_meld_startindex + 16] := FALSE;
	garr_stoermeldungen[st_config.i16_meld_startindex + 17] := FALSE;
	garr_stoermeldungen[st_config.i16_meld_startindex + 18] := FALSE;
	garr_stoermeldungen[st_config.i16_meld_startindex + 19] := FALSE;
	
	garr_betriebsmeldungen[st_config.i16_meld_startindex + 0] := bm_setze_anforderung;
	garr_betriebsmeldungen[st_config.i16_meld_startindex + 1] := bm_abfrage_wt_an_stopper;
	garr_betriebsmeldungen[st_config.i16_meld_startindex + 2] := FALSE;
	garr_betriebsmeldungen[st_config.i16_meld_startindex + 3] := FALSE;
	garr_betriebsmeldungen[st_config.i16_meld_startindex + 4] := FALSE;
	garr_betriebsmeldungen[st_config.i16_meld_startindex + 5] := FALSE;
	garr_betriebsmeldungen[st_config.i16_meld_startindex + 6] := FALSE;
	garr_betriebsmeldungen[st_config.i16_meld_startindex + 7] := FALSE;
	garr_betriebsmeldungen[st_config.i16_meld_startindex + 8] := FALSE;
	garr_betriebsmeldungen[st_config.i16_meld_startindex + 9] := FALSE;
	garr_betriebsmeldungen[st_config.i16_meld_startindex + 10] := FALSE;
	garr_betriebsmeldungen[st_config.i16_meld_startindex + 11] := FALSE;
	garr_betriebsmeldungen[st_config.i16_meld_startindex + 12] := FALSE;
	garr_betriebsmeldungen[st_config.i16_meld_startindex + 13] := FALSE;
	garr_betriebsmeldungen[st_config.i16_meld_startindex + 14] := FALSE;
	garr_betriebsmeldungen[st_config.i16_meld_startindex + 15] := FALSE;
	garr_betriebsmeldungen[st_config.i16_meld_startindex + 16] := FALSE;
	garr_betriebsmeldungen[st_config.i16_meld_startindex + 17] := FALSE;
	garr_betriebsmeldungen[st_config.i16_meld_startindex + 18] := FALSE;
	garr_betriebsmeldungen[st_config.i16_meld_startindex + 19] := FALSE;
END_IF
END_PROGRAM

(* POU Gemeinsamkeiten17xx/WT Transport/ST_Hublift_rechts, ST *)
PROGRAM ST_Hublift_rechts
VAR_INPUT
	st_config							: struct_config;
	st_ctrl_in							: struct_ctrl_in;
	e_station_vorher_in_anforderung		: BOOL := FALSE;
	e_station_vorher_in_abgegeben		: BOOL := FALSE;
END_VAR
VAR_IN_OUT
	st_visu							: struct_visu;
END_VAR
VAR_OUTPUT
	st_ctrl_out						: struct_ctrl_out;
	a_station_vorher_out_erlaubnis		: BOOL := FALSE;
	a_station_vorher_out_angekommen	: BOOL := FALSE;
END_VAR
VAR
	fb_ton_wz						: TON;
	fb_ton_uez						: TON;
	fb_ton_quitt						: TON;
	fb_ton_wt_anwesend			: TON;
	fb_state_entry					: ST_StateEntry;
	sm_kein_wt_anwesend			: BOOL := FALSE;
	sm_kein_wt_eingeklinkt			: BOOL := FALSE;
	sm_keine_busverbindung		: BOOL := FALSE;

	e_sensor_wt_anwesend			AT %I* : BOOL;
	e_wc_state						AT%I*: BOOL;	(* 0=Data valid, 1=Data invalid *)
END_VAR
(* Zeiten *)
fb_ton_wz(IN:= , PT:= , Q=>  , ET=> );
fb_ton_uez(IN:= , PT:= , Q=>  , ET=> );
fb_ton_quitt(IN:= , PT:= t#100ms, Q=> , ET=> );
fb_ton_wt_anwesend(IN:= e_sensor_wt_anwesend, PT:= t#200ms, Q=> , ET=> );

(* Toplevel *)
IF fb_state_entry.i16_next_step > INIT AND fb_state_entry.i16_next_step < FEHLER THEN
	IF fb_state_entry.i16_next_step < STOP THEN
		IF st_ctrl_in.b_stop THEN
			fb_state_entry.i16_next_step := STOP;
		END_IF
	END_IF

	(* Allgemeine Fehler *)
	IF 	st_config.b_station_aktiv AND NOT st_config.b_station_in_simulation AND
		(zyl_hublift_rechts_lift.st_ctrl.out.b_fehler OR
		zyl_hublift_rechts_wt_einzug.st_ctrl.out.b_fehler OR
		zyl_hublift_rechts_wt_klinke.st_ctrl.out.b_fehler)
		THEN
			fb_state_entry.i16_next_step := FEHLER;

	(* Zylinder im Handbetrieb *)
	ELSIF gi16_betriebsart = HAND AND st_config.b_station_aktiv AND NOT st_config.b_station_in_simulation AND
		((st_visu.st_zyl.i16_nr_zyl_im_handbetrieb = zyl_hublift_rechts_lift.fb.st_config.i16_identnummer) OR
		(st_visu.st_zyl.i16_nr_zyl_im_handbetrieb = zyl_hublift_rechts_wt_einzug.fb.st_config.i16_identnummer) OR
		(st_visu.st_zyl.i16_nr_zyl_im_handbetrieb = zyl_hublift_rechts_wt_klinke.fb.st_config.i16_identnummer))
		THEN
			fb_state_entry.i16_next_step := FEHLER;
	END_IF
END_IF

(* ==================================Schrittkette================================ *)
fb_state_entry(
	i16_next_step:= , 
	i16_pos:= 1,
	s_debugtext:= ,
	E=> ,
	X=> , 
	i16_step=> ,
	i16_last_step=> );

CASE fb_state_entry.i16_step OF
(*=======================================================*)
	INIT_OBJ:
		IF st_config.b_config_fertig THEN
			fb_state_entry.i16_next_step := INIT;
		END_IF

(*=======================================================*)
	INIT:
		IF fb_state_entry.E THEN
			fb_ton_wz.IN := FALSE;
			fb_ton_uez.IN	:= FALSE;
			fb_ton_quitt.IN := FALSE;
			sm_kein_wt_anwesend	:= FALSE;
			sm_kein_wt_eingeklinkt := FALSE;
			sm_keine_busverbindung := FALSE;
			a_station_vorher_out_erlaubnis := FALSE;
			a_station_vorher_out_angekommen := FALSE;
			st_ctrl_out.b_fehler := FALSE;
			st_ctrl_out.b_bereit := FALSE;
			st_ctrl_out.b_fertig := FALSE;
			zyl_hublift_rechts_lift.st_ctrl.in.b_einfahren := FALSE;
			zyl_hublift_rechts_lift.st_ctrl.in.b_ausfahren := FALSE;
			zyl_hublift_rechts_wt_einzug.st_ctrl.in.b_einfahren := FALSE;
			zyl_hublift_rechts_wt_einzug.st_ctrl.in.b_ausfahren := FALSE;
			zyl_hublift_rechts_wt_klinke.st_ctrl.in.b_einfahren := FALSE;
			zyl_hublift_rechts_wt_klinke.st_ctrl.in.b_ausfahren := FALSE;
		END_IF

		(*-----------------------Weiterschaltbedingungen----------------------------*)
		IF st_ctrl_in.b_init THEN
			zyl_hublift_rechts_lift.st_ctrl.in.b_quittieren := FALSE;
			zyl_hublift_rechts_wt_einzug.st_ctrl.in.b_quittieren := FALSE;
			zyl_hublift_rechts_wt_klinke.st_ctrl.in.b_quittieren := FALSE;
			IF	 st_config.b_station_aktiv AND NOT st_config.b_station_in_simulation AND
				(gst_datensatz.st_md.b_wt_transport_aktiv OR gst_datensatz.st_md.b_wt_transport_simulation) THEN
					fb_state_entry.i16_next_step := 15;
			ELSE
				fb_state_entry.i16_next_step := BEREIT;
			END_IF
		END_IF

(*=======================================================*)
	15: (* Prüfe, ob Busverbindung vorhanden ist *)

		(*-----------------------Weiterschaltbedingungen----------------------------*)
		IF 	zyl_hublift_rechts_lift.fb.e_sensor1_ausgefahren OR
			zyl_hublift_rechts_lift.fb.e_sensor1_eingefahren OR
			zyl_hublift_rechts_wt_einzug.fb.e_sensor1_ausgefahren OR
			zyl_hublift_rechts_wt_einzug.fb.e_sensor1_eingefahren OR
			zyl_hublift_rechts_wt_klinke.fb.e_sensor1_ausgefahren OR
			zyl_hublift_rechts_wt_klinke.fb.e_sensor1_eingefahren THEN
				fb_state_entry.i16_next_step := 20;
		ELSE
				sm_keine_busverbindung := TRUE;
				fb_state_entry.i16_next_step := FEHLER;
		END_IF


		(* Bei der nächsten TSM Änderung bitte aktivieren
		IF e_wc_state THEN
			sm_keine_busverbindung := TRUE;
			fb_state_entry.i16_next_step := FEHLER;
		ELSE
			fb_state_entry.i16_next_step := 20;
		END_IF*)

(*=======================================================*)
	20: (* Initialisierung: Prüfe WT in Lift *)

		(*-----------------------Weiterschaltbedingungen----------------------------*)
		IF fb_ton_wt_anwesend.Q  THEN
			(* WT ist angekommen *)
			fb_state_entry.i16_next_step := 50;
		ELSE
			fb_state_entry.i16_next_step := 30;
		END_IF

(*=======================================================*)
	30: (* Initialisierung: Klinke einfahren *)
		IF fb_state_entry.E THEN
			zyl_hublift_rechts_wt_klinke.st_ctrl.in.b_einfahren := TRUE;
		END_IF

		(*-----------------------Weiterschaltbedingungen----------------------------*)
		IF zyl_hublift_rechts_wt_klinke.st_ctrl.out.b_eingefahren THEN
			zyl_hublift_rechts_wt_klinke.st_ctrl.in.b_einfahren := FALSE;
			fb_state_entry.i16_next_step := 35;
		END_IF

(*=======================================================*)
	35: (* Initialisierung: WT-Einzug einfahren *)
		IF fb_state_entry.E THEN
			zyl_hublift_rechts_wt_einzug.st_ctrl.in.b_einfahren := TRUE;
		END_IF

		(*-----------------------Weiterschaltbedingungen----------------------------*)
		IF zyl_hublift_rechts_wt_einzug.st_ctrl.out.b_eingefahren THEN
			zyl_hublift_rechts_wt_einzug.st_ctrl.in.b_einfahren := FALSE;
			fb_state_entry.i16_next_step := 40;
		END_IF

(*=======================================================*)
	40: (* Initialisierung: Lift Hoch *)
		IF fb_state_entry.E THEN
			zyl_hublift_rechts_lift.st_ctrl.in.b_ausfahren := TRUE;
		END_IF

		(*-----------------------Weiterschaltbedingungen----------------------------*)
		IF zyl_hublift_rechts_lift.st_ctrl.out.b_ausgefahren THEN
			zyl_hublift_rechts_lift.st_ctrl.in.b_ausfahren := FALSE;
			fb_state_entry.i16_next_step := 45;
		END_IF

(*=======================================================*)
	45: (* Initialisierung: WT-Einzug ausfahren *)
		IF fb_state_entry.E THEN
			zyl_hublift_rechts_wt_einzug.st_ctrl.in.b_ausfahren := TRUE;
		END_IF

		(*-----------------------Weiterschaltbedingungen----------------------------*)
		IF zyl_hublift_rechts_wt_einzug.st_ctrl.out.b_ausgefahren THEN
			zyl_hublift_rechts_wt_einzug.st_ctrl.in.b_ausfahren := FALSE;
			fb_state_entry.i16_next_step := BEREIT;
		END_IF

(*=======================================================*)
	50: (* Initialisierung: Klinke ausfahren *)
		IF fb_state_entry.E THEN
			zyl_hublift_rechts_wt_klinke.st_ctrl.in.b_ausfahren := TRUE;
		END_IF

		(*-----------------------Weiterschaltbedingungen----------------------------*)
		IF zyl_hublift_rechts_wt_klinke.st_ctrl.out.b_ausgefahren THEN
			zyl_hublift_rechts_wt_klinke.st_ctrl.in.b_ausfahren := FALSE;
			fb_state_entry.i16_next_step := 55;
		END_IF

(*=======================================================*)
	55: (* Initialisierung: WT-Einzug einfahren *)
		IF fb_state_entry.E THEN
			zyl_hublift_rechts_wt_einzug.st_ctrl.in.b_einfahren := TRUE;
		END_IF

		(*-----------------------Weiterschaltbedingungen----------------------------*)
		IF zyl_hublift_rechts_wt_einzug.st_ctrl.out.b_eingefahren THEN
			zyl_hublift_rechts_wt_einzug.st_ctrl.in.b_einfahren := FALSE;
			fb_state_entry.i16_next_step := 60;
		END_IF

(*=======================================================*)
	60: (* Initialisierung: Lift einfahren *)
		IF fb_state_entry.E THEN
			zyl_hublift_rechts_lift.st_ctrl.in.b_einfahren := TRUE;
		END_IF

		(*-----------------------Weiterschaltbedingungen----------------------------*)
		IF zyl_hublift_rechts_lift.st_ctrl.out.b_eingefahren THEN
			zyl_hublift_rechts_lift.st_ctrl.in.b_einfahren := FALSE;
			fb_state_entry.i16_next_step := 65;
		END_IF

(*=======================================================*)
	65: (* Initialisierung: WT-Einzug ausfahren *)
		IF fb_state_entry.E THEN
			zyl_hublift_rechts_wt_einzug.st_ctrl.in.b_ausfahren := TRUE;
		END_IF

		(*-----------------------Weiterschaltbedingungen----------------------------*)
		IF zyl_hublift_rechts_wt_einzug.st_ctrl.out.b_ausgefahren THEN
			zyl_hublift_rechts_wt_einzug.st_ctrl.in.b_ausfahren := FALSE;
			fb_state_entry.i16_next_step := 70;
		END_IF

(*=======================================================*)
	70: (* Initialisierung: Klinke einfahren *)
		IF fb_state_entry.E THEN
			zyl_hublift_rechts_wt_klinke.st_ctrl.in.b_einfahren := TRUE;
		END_IF

		(*-----------------------Weiterschaltbedingungen----------------------------*)
		IF zyl_hublift_rechts_wt_klinke.st_ctrl.out.b_eingefahren THEN
			zyl_hublift_rechts_wt_klinke.st_ctrl.in.b_einfahren := FALSE;
			fb_state_entry.i16_next_step := 75;
		END_IF

(*=======================================================*)
	75: (* Initialisierung: Warte WT vom Förderband eingezogen *)
		IF fb_state_entry.E THEN
			fb_ton_wz.PT :=t#300ms;
			fb_ton_wz.IN := TRUE;
		END_IF

		(*-----------------------Weiterschaltbedingungen----------------------------*)
		IF fb_ton_wz.Q THEN
			fb_ton_wz.IN := FALSE;
			fb_state_entry.i16_next_step := 80;
		END_IF

(*=======================================================*)
	80: (* Initialisierung: WT-Einzug einfahren *)
		IF fb_state_entry.E THEN
			zyl_hublift_rechts_wt_einzug.st_ctrl.in.b_einfahren := TRUE;
		END_IF

		(*-----------------------Weiterschaltbedingungen----------------------------*)
		IF zyl_hublift_rechts_wt_einzug.st_ctrl.out.b_eingefahren THEN
			zyl_hublift_rechts_wt_einzug.st_ctrl.in.b_einfahren := FALSE;
			fb_state_entry.i16_next_step := 85;
		END_IF

(*=======================================================*)
	85: (* Initialisierung: Lift Hoch *)
		IF fb_state_entry.E THEN
			zyl_hublift_rechts_lift.st_ctrl.in.b_ausfahren := TRUE;
		END_IF

		(*-----------------------Weiterschaltbedingungen----------------------------*)
		IF zyl_hublift_rechts_lift.st_ctrl.out.b_ausgefahren THEN
			zyl_hublift_rechts_lift.st_ctrl.in.b_ausfahren := FALSE;
			fb_state_entry.i16_next_step := 90;
		END_IF

(*=======================================================*)
	90: (* Initialisierung: WT-Einzug ausfahren *)
		IF fb_state_entry.E THEN
			zyl_hublift_rechts_wt_einzug.st_ctrl.in.b_ausfahren := TRUE;
		END_IF

		(*-----------------------Weiterschaltbedingungen----------------------------*)
		IF zyl_hublift_rechts_wt_einzug.st_ctrl.out.b_ausgefahren THEN
			zyl_hublift_rechts_wt_einzug.st_ctrl.in.b_ausfahren := FALSE;
			a_station_vorher_out_angekommen := TRUE;	(* benötigtes Signal, damit es an der Vorgängerzelle in "ST_WT_Transport_Abgabe" weiter gehen kann *)
			fb_state_entry.i16_next_step := BEREIT;
		END_IF

(*=======================================================*)
	BEREIT:	(* Warte auf Anforderung von vorheriger Station zum aufnehmen des WT *)
		IF fb_state_entry.E THEN
			a_station_vorher_out_erlaubnis := FALSE;
			st_ctrl_out.b_bereit := TRUE;
		END_IF

		(*-----------------------Weiterschaltbedingungen----------------------------*)
		IF 	(st_config.b_station_aktiv OR st_config.b_station_in_simulation) AND
			(gst_datensatz.st_md.b_wt_transport_aktiv OR gst_datensatz.st_md.b_wt_transport_simulation)
			THEN
				(* Hublift und WT Transport aktiv - die Simulation spielt im weiteren Verlauf keine Rolle mehr *)
				IF e_station_vorher_in_anforderung THEN
					a_station_vorher_out_angekommen := FALSE;
					a_station_vorher_out_erlaubnis := TRUE;
					fb_state_entry.i16_next_step := 120;
				END_IF
		ELSE
			;(* Hublift und WT Transport NICHT aktiv *)
		END_IF

(*=======================================================*)
	110: (* Warte bis WT abgegeben wurde*)
		IF fb_state_entry.E THEN
			a_station_vorher_out_erlaubnis := TRUE;
		END_IF

		(*-----------------------Weiterschaltbedingungen----------------------------*)
		IF e_station_vorher_in_abgegeben AND NOT fb_state_entry.E THEN
			a_station_vorher_out_erlaubnis := FALSE;
			fb_state_entry.i16_next_step := 120;
		END_IF

(*=======================================================*)
	120:	(* Abfrage, ob der WT auch eingehakt wurde *)
		IF fb_state_entry.E THEN
			fb_ton_wz.PT := t#2s;
			fb_ton_wz.IN := TRUE;
		END_IF

		(*-----------------------Weiterschaltbedingungen----------------------------*)
		IF fb_ton_wt_anwesend.Q  THEN
			(* WT ist angekommen *)
			fb_ton_wz.IN := FALSE;
			fb_state_entry.i16_next_step := 130;
		END_IF

		(* Pfad für nicht angekommen oder Simulation *)
		IF fb_ton_wz.Q THEN
			a_station_vorher_out_angekommen := TRUE;
			fb_ton_wz.IN := FALSE;
			fb_state_entry.i16_next_step := BEREIT;
		END_IF

(*=======================================================*)
	130: (* Klinke ausfahren -> WT einhaken*)
		IF fb_state_entry.E THEN
			zyl_hublift_rechts_wt_klinke.st_ctrl.in.b_ausfahren := TRUE;
		END_IF

		(*-----------------------Weiterschaltbedingungen----------------------------*)
		IF zyl_hublift_rechts_wt_klinke.st_ctrl.out.b_ausgefahren AND gb_ba_auto_kontroller THEN
			zyl_hublift_rechts_wt_klinke.st_ctrl.in.b_ausfahren := FALSE;
			fb_state_entry.i16_next_step := 140;
		END_IF

(*=======================================================*)
	140: (* WT-Einzug einfahren *)
		IF fb_state_entry.E THEN
			zyl_hublift_rechts_wt_einzug.st_ctrl.in.b_einfahren := TRUE;
		END_IF

		(*-----------------------Weiterschaltbedingungen----------------------------*)
		IF zyl_hublift_rechts_wt_einzug.st_ctrl.out.b_eingefahren AND gb_ba_auto_kontroller THEN
			zyl_hublift_rechts_wt_einzug.st_ctrl.in.b_einfahren := FALSE;
			IF e_sensor_wt_anwesend THEN
				a_station_vorher_out_erlaubnis := FALSE;
				a_station_vorher_out_angekommen := TRUE;
				fb_state_entry.i16_next_step := 150;
			ELSE
				sm_kein_wt_eingeklinkt := TRUE;
				fb_state_entry.i16_next_step := FEHLER;
			END_IF
		END_IF

(*=======================================================*)
	150: (* WT mit Lift absenken *)
		IF fb_state_entry.E THEN
			zyl_hublift_rechts_lift.st_ctrl.in.b_einfahren := TRUE;
		END_IF

		(*-----------------------Weiterschaltbedingungen----------------------------*)
		IF zyl_hublift_rechts_lift.st_ctrl.out.b_eingefahren AND gb_ba_auto_kontroller THEN
			zyl_hublift_rechts_lift.st_ctrl.in.b_einfahren := FALSE;
			fb_state_entry.i16_next_step := 160;
		END_IF

(*=======================================================*)
	160: (* WT-Einzug ausfahren und Klinke einfahren und WT aushaken*)
		IF fb_state_entry.E THEN
			zyl_hublift_rechts_wt_einzug.st_ctrl.in.b_ausfahren := TRUE;
			zyl_hublift_rechts_wt_klinke.st_ctrl.in.b_einfahren := TRUE;
		END_IF

		(*-----------------------Weiterschaltbedingungen----------------------------*)
		IF 	zyl_hublift_rechts_wt_einzug.st_ctrl.out.b_ausgefahren AND
			zyl_hublift_rechts_wt_klinke.st_ctrl.out.b_eingefahren AND
			gb_ba_auto_kontroller
			THEN
				zyl_hublift_rechts_wt_einzug.st_ctrl.in.b_ausfahren := FALSE;
				zyl_hublift_rechts_wt_klinke.st_ctrl.in.b_einfahren := FALSE;
				fb_state_entry.i16_next_step := 170;
		END_IF

(*=======================================================*)
	170:	(* WT wird von FB reingezogen *)

		(*-----------------------Weiterschaltbedingungen----------------------------*)
		IF NOT e_sensor_wt_anwesend THEN;
			fb_ton_wz.PT := t#500ms;
			fb_ton_wz.IN := TRUE;
			IF fb_ton_wz.Q THEN
				fb_ton_wz.IN := FALSE;
				fb_state_entry.i16_next_step := 180;
			END_IF
		END_IF

(*=======================================================*)
	180: (* Lift ausfahren *)
		IF fb_state_entry.E THEN
			zyl_hublift_rechts_lift.st_ctrl.in.b_ausfahren := TRUE;
		END_IF

		(*-----------------------Weiterschaltbedingungen----------------------------*)
		IF zyl_hublift_rechts_lift.st_ctrl.out.b_ausgefahren THEN
			zyl_hublift_rechts_lift.st_ctrl.in.b_ausfahren := FALSE;
			fb_state_entry.i16_next_step := BEREIT;
		END_IF

(*=======================================================*)
	FEHLER:
		IF fb_state_entry.E THEN
			fb_ton_quitt.IN := FALSE;
			st_ctrl_out.b_fehler := TRUE;
			a_station_vorher_out_erlaubnis := FALSE;
			a_station_vorher_out_angekommen := FALSE;
			zyl_hublift_rechts_lift.st_ctrl.in.b_quittieren := FALSE;
			zyl_hublift_rechts_wt_einzug.st_ctrl.in.b_quittieren := FALSE;
			zyl_hublift_rechts_wt_klinke.st_ctrl.in.b_quittieren := FALSE;
		END_IF

		(*-----------------------Weiterschaltbedingungen----------------------------*)
		IF st_ctrl_in.b_quitt AND NOT fb_state_entry.E THEN
			st_ctrl_out.b_fehler := FALSE;
			zyl_hublift_rechts_lift.st_ctrl.in.b_quittieren := TRUE;
			zyl_hublift_rechts_wt_einzug.st_ctrl.in.b_quittieren := TRUE;
			zyl_hublift_rechts_wt_klinke.st_ctrl.in.b_quittieren := TRUE;
			fb_ton_quitt.IN := TRUE;
		END_IF

		IF fb_ton_quitt.Q THEN
			fb_ton_quitt.IN := FALSE;
			fb_state_entry.i16_next_step := INIT;
		END_IF

(*=======================================================*)
	STOP:
		IF fb_state_entry.E THEN
			fb_ton_quitt.IN := FALSE;
			zyl_hublift_rechts_lift.st_ctrl.in.b_quittieren := FALSE;
			zyl_hublift_rechts_wt_einzug.st_ctrl.in.b_quittieren := FALSE;
			zyl_hublift_rechts_wt_klinke.st_ctrl.in.b_quittieren := FALSE;
		END_IF

		(*-----------------------Weiterschaltbedingungen----------------------------*)
		IF st_ctrl_in.b_quitt AND NOT fb_state_entry.E THEN
			fb_ton_quitt.IN := TRUE;
			zyl_hublift_rechts_lift.st_ctrl.in.b_quittieren := TRUE;
			zyl_hublift_rechts_wt_einzug.st_ctrl.in.b_quittieren := TRUE;
			zyl_hublift_rechts_wt_klinke.st_ctrl.in.b_quittieren := TRUE;
		END_IF

		IF fb_ton_quitt.Q THEN
			fb_ton_quitt.IN := FALSE;
			fb_state_entry.i16_next_step := INIT;
		END_IF
END_CASE


fb_state_entry(
	i16_next_step:= , 
	i16_pos:= 2,
	s_debugtext:= ,
	E=> , 
	X=> ,
	i16_step=> ,
	i16_last_step=> );

IF st_config.b_config_fertig THEN
	(* Fehlermeldungen und Betriebsmeldungen ab dem Startindex in die globalen Meldungsarrays schreiben *)
	garr_stoermeldungen[st_config.i16_meld_startindex + 0] := sm_kein_wt_anwesend;
	garr_stoermeldungen[st_config.i16_meld_startindex + 1] := sm_kein_wt_eingeklinkt;
	garr_stoermeldungen[st_config.i16_meld_startindex + 2] := sm_keine_busverbindung;
	garr_stoermeldungen[st_config.i16_meld_startindex + 3] := FALSE;
	garr_stoermeldungen[st_config.i16_meld_startindex + 4] := FALSE;
	garr_stoermeldungen[st_config.i16_meld_startindex + 5] := FALSE;
	garr_stoermeldungen[st_config.i16_meld_startindex + 6] := FALSE;
	garr_stoermeldungen[st_config.i16_meld_startindex + 7] := FALSE;
	garr_stoermeldungen[st_config.i16_meld_startindex + 8] := FALSE;
	garr_stoermeldungen[st_config.i16_meld_startindex + 9] := FALSE;
	garr_stoermeldungen[st_config.i16_meld_startindex + 10] := FALSE;
	garr_stoermeldungen[st_config.i16_meld_startindex + 11] := FALSE;
	garr_stoermeldungen[st_config.i16_meld_startindex + 12] := FALSE;
	garr_stoermeldungen[st_config.i16_meld_startindex + 13] := FALSE;
	garr_stoermeldungen[st_config.i16_meld_startindex + 14] := FALSE;
	garr_stoermeldungen[st_config.i16_meld_startindex + 15] := FALSE;
	garr_stoermeldungen[st_config.i16_meld_startindex + 16] := FALSE;
	garr_stoermeldungen[st_config.i16_meld_startindex + 17] := FALSE;
	garr_stoermeldungen[st_config.i16_meld_startindex + 18] := FALSE;
	garr_stoermeldungen[st_config.i16_meld_startindex + 19] := FALSE;
	
	garr_betriebsmeldungen[st_config.i16_meld_startindex + 0] := FALSE;
	garr_betriebsmeldungen[st_config.i16_meld_startindex + 1] := FALSE;
	garr_betriebsmeldungen[st_config.i16_meld_startindex + 2] := FALSE;
	garr_betriebsmeldungen[st_config.i16_meld_startindex + 3] := FALSE;
	garr_betriebsmeldungen[st_config.i16_meld_startindex + 4] := FALSE;
	garr_betriebsmeldungen[st_config.i16_meld_startindex + 5] := FALSE;
	garr_betriebsmeldungen[st_config.i16_meld_startindex + 6] := FALSE;
	garr_betriebsmeldungen[st_config.i16_meld_startindex + 7] := FALSE;
	garr_betriebsmeldungen[st_config.i16_meld_startindex + 8] := FALSE;
	garr_betriebsmeldungen[st_config.i16_meld_startindex + 9] := FALSE;
	garr_betriebsmeldungen[st_config.i16_meld_startindex + 10] := FALSE;
	garr_betriebsmeldungen[st_config.i16_meld_startindex + 11] := FALSE;
	garr_betriebsmeldungen[st_config.i16_meld_startindex + 12] := FALSE;
	garr_betriebsmeldungen[st_config.i16_meld_startindex + 13] := FALSE;
	garr_betriebsmeldungen[st_config.i16_meld_startindex + 14] := FALSE;
	garr_betriebsmeldungen[st_config.i16_meld_startindex + 15] := FALSE;
	garr_betriebsmeldungen[st_config.i16_meld_startindex + 16] := FALSE;
	garr_betriebsmeldungen[st_config.i16_meld_startindex + 17] := FALSE;
	garr_betriebsmeldungen[st_config.i16_meld_startindex + 18] := FALSE;
	garr_betriebsmeldungen[st_config.i16_meld_startindex + 19] := FALSE;
END_IF
END_PROGRAM

(* POU Maschine1700/WT Transport/ST_WT_Transport_Beladen, ST *)
PROGRAM ST_WT_Transport_Beladen
VAR_INPUT
	st_config								: struct_config;
	st_ctrl_in								: struct_ctrl_in;
	e_station_vorher_in_anforderung			: BOOL := FALSE;
	e_station_vorher_in_abgegeben			: BOOL := FALSE;
END_VAR
VAR_IN_OUT
	st_visu								: struct_visu;
END_VAR
VAR_OUTPUT
	st_ctrl_out							: struct_ctrl_out;
	a_station_vorher_out_erlaubnis			: BOOL := FALSE;
	a_station_vorher_out_angekommen		: BOOL := FALSE;
	t_WT_WechselZeit					: TIME := t#0ms;
	t_traegerwechselzeit					: TIME := t#0ms;
	t_Zentrierer_ausfahren					: TIME := t#0ms;
	t_Zentrierer_einfahren					: TIME := t#0ms;
	t_komplett_zyklus						: TIME := t#0ms;
END_VAR
VAR
	fb_ton_uez							: TON;
	fb_ton_wz							: TON;
	fb_ton_quitt							: TON;
	fb_ton_wt_auf_beladepos				: TON;
	fb_tof_wt_auf_beladepos				: TOF;
	fb_r_trig_start							: R_TRIG;
	fb_r_trig_beladepos					: R_TRIG;
	fb_r_trig_beladepos_verlassen			: R_TRIG;
	fb_r_trig_pm_time						: R_TRIG;
	fb_state_entry							: ST_StateEntry;
	sm_wt_hat_beladepos_nicht_verlassen	: BOOL := FALSE;
	sm_tagnummer_ungueltig				: BOOL := FALSE;
	sm_wt_hat_kein_tag					: BOOL := FALSE;
	sm_tagreader_nicht_fertig				: BOOL := FALSE;
	sm_wt_zu_frueh_in_zelle				: BOOL := FALSE;
	sm_keine_bandfreigabe				: BOOL := FALSE;
	bm_abfrage_wt_auf_beladepos			: BOOL := FALSE;
	bm_warte_anforderung					: BOOL := FALSE;
	bm_warte_auf_wt_an_stopper			: BOOL := FALSE;
	bMerkerSchrittketteKommtVonInit		: BOOL := FALSE;
	fb_ton_abfrage_wt_auf_beladepos		: TON;
	fb_ton_warte_anforderung				: TON;
	fb_ton_warte_auf_wt_an_stopper			: TON;
	fb_WT_WechselZeit					: ST_Taktzeit;
	fb_Tisch_WechselZeit					: ST_Taktzeit;
	fb_Zentrierer_ausfahren				: ST_Taktzeit;
	fb_Zentrierer_einfahren					: ST_Taktzeit;
	t_bestueckzeit						: TIME := t#0ms;
	i									: INT := 0;

	sm_sensorfehler_beladepos			: BOOL := FALSE;

	(* zum Testen der Achsen nach Tausch, Bestückbild "Becherspucken", WKZ ausgebaut, Vorschubkontrolle abeschaltet,
	Bit muss von Programmierer geforct werden, zum Beenden Schlüsselschalter auf HAND und Zelle neu starten *)
	b_Dauertest_Achsen					: BOOL := FALSE;

	e_wt_auf_beladepos					AT %I* : BOOL;
	e_wt_im_aktionsfeld					AT %I* : BOOL;
	e_wt_beladepos_verlassen				AT %I* : BOOL;
	e_wt_auf_pufferstrecke					AT %I* : BOOL;
	e_wt_faellt_in_achse_ueberw			AT %I* : BOOL;

	zeit_wt_kompletter_zyklus				: DINT := 0;

	i16_state_msg						: INT;
	pm_traegerwechselzeit					: BOOL := FALSE;
	t_tischwechselzeit					: TIME := t#0ms;
	t_tischwechselzeit_help				: TIME := t#0ms;

END_VAR
(* Zeiten *)
fb_ton_uez(IN:= , PT:= , Q=>  , ET=> );
fb_ton_wz(IN:= , PT:= , Q=> , ET=> );
fb_ton_quitt(IN:= , PT:= t#100ms, Q=> , ET=> );

fb_ton_wt_auf_beladepos(IN:= e_wt_auf_beladepos, PT:= t#100ms, Q=> , ET=> );
fb_tof_wt_auf_beladepos(IN:= e_wt_auf_beladepos, PT:= t#100ms, Q=> , ET=> );

(* Flanken *)
fb_r_trig_beladepos(CLK:= e_wt_auf_beladepos, Q=> );
fb_r_trig_beladepos_verlassen(CLK:= e_wt_beladepos_verlassen, Q=> );
fb_r_trig_start(CLK:= st_ctrl_in.b_start, Q=> );

(*Trägerwechselzeiten*)
fb_WT_WechselZeit(b_start:= , t_zeit=> );
fb_Zentrierer_ausfahren(b_start:= , t_zeit=> );
fb_Zentrierer_einfahren(b_start:= , t_zeit=> );
fb_Tisch_WechselZeit(b_start:= , t_zeit=> );


(*Meldung für Trägerwechselzeit zu groß*)
fb_r_trig_pm_time(CLK:= pm_traegerwechselzeit, Q=> );

IF fb_r_trig_pm_time.Q  THEN
	t_tischwechselzeit_help := t_tischwechselzeit;
	i16_state_msg := 1;
END_IF

(*Produktionsmeldung für Übergabe zu lange*)
CASE i16_state_msg OF
	1: (*Warten bis keine ander Produktions Meldung ansteht *)
		IF	TestAndSet(ST_Message_Produktion.LockFlag) THEN
			ST_Message_Produktion.ClearMessageLines();
			i16_state_msg := 2;
		END_IF

	2:  (*Produktions Meldung*)
		Visu.MeldungProduktion.Color_R := 255;
		Visu.MeldungProduktion.Color_G := 255;
		Visu.MeldungProduktion.Color_B := 0;
		IF visu.s_akt_sprache = 'de' THEN
			Visu.MeldungProduktion.Name:=CONCAT('WT zu langsam vom Tisch gefahren.',TIME_TO_STRING(t_tischwechselzeit_help));
		ELSIF visu.s_akt_sprache = 'en' THEN
			Visu.MeldungProduktion.Name:=CONCAT('carrier exceeded time to leave stiching table.',TIME_TO_STRING(t_tischwechselzeit_help));
		ELSIF visu.s_akt_sprache = 'cz' THEN
			Visu.MeldungProduktion.Name:=CONCAT('Prekroceni casu vyjezdu paletky z osazovani.',TIME_TO_STRING(t_tischwechselzeit_help));
		END_IF
		Visu.MeldungProduktion.ShowMessage := TRUE;
		Visu.MeldungProduktion.Button1.sichtbar:=TRUE;	(*OK*)
		Visu.MeldungProduktion.Button1.Text:='Ok';
		i16_state_msg := 3;

	3:  (*Warte auf OK*)
		IF Visu.MeldungProduktion.Button1.tasten THEN
			i16_state_msg:=0;
		END_IF
END_CASE

(* ==================================Toplevel=================================== *)
IF fb_state_entry.i16_next_step > INIT AND fb_state_entry.i16_next_step < FEHLER THEN
	IF st_ctrl_in.b_stop THEN
		fb_state_entry.i16_next_step := STOP;

	(* Allgemeine Fehler *)
	ELSIF zyl_wt_zentrierer_tisch.st_ctrl.out.b_fehler OR zyl_wt_stopper_tisch.st_ctrl.out.b_fehler THEN
		fb_state_entry.i16_next_step := FEHLER;

	(* Überwachung ob ein WT zu früh in die Zelle fällt und dadurch die Z-Achse beschädigt *)
	ELSIF e_wt_faellt_in_achse_ueberw AND ST_Z_Achse.fb_state_entry.i16_step >=130 AND
		ST_Z_Achse.fb_state_entry.i16_step < FEHLER THEN
			sm_wt_zu_frueh_in_zelle := TRUE;
			fb_state_entry.i16_next_step := FEHLER;

	(* Zylinder im Handbetrieb *)
	ELSIF gi16_betriebsart = HAND AND
		(st_visu.st_zyl.i16_nr_zyl_im_handbetrieb = zyl_wt_zentrierer_tisch.fb.st_config.i16_identnummer OR
		st_visu.st_zyl.i16_nr_zyl_im_handbetrieb = zyl_wt_stopper_tisch.fb.st_config.i16_identnummer)
		THEN
			fb_state_entry.i16_next_step := FEHLER;
	END_IF
END_IF

(* ============================Haupt-Schrittkette================================ *)
fb_state_entry(
	i16_next_step:= ,
	i16_pos:= 1,
	s_debugtext:= ,
	E=> ,
	X=> , 
	i16_step=> ,
	i16_last_step=> );

CASE fb_state_entry.i16_step OF
(*=======================================================*)
	INIT_OBJ:
		IF st_config.b_config_fertig THEN
			fb_state_entry.i16_next_step := INIT;
		END_IF

(*=======================================================*)
	INIT:
		IF fb_state_entry.E THEN
			fb_ton_wz.IN := FALSE;
			fb_ton_uez.IN := FALSE;
			fb_ton_quitt.IN := FALSE;
			st_ctrl_out.b_fehler := FALSE;
			st_ctrl_out.b_bereit := FALSE;
			st_ctrl_out.b_fertig := FALSE;
			st_ctrl_out.b_kontroller_start := FALSE;
			zyl_wt_zentrierer_tisch.st_ctrl.in.b_einfahren := FALSE;
			zyl_wt_zentrierer_tisch.st_ctrl.in.b_ausfahren := TRUE;
			zyl_wt_stopper_tisch.st_ctrl.in.b_einfahren := FALSE;
			zyl_wt_stopper_tisch.st_ctrl.in.b_ausfahren := FALSE;
			axis_z_achse.st_ctrl.in.b_start := FALSE;
			stueckzahlen.st_ctrl.in.b_gutteil_produziert := FALSE;
			sm_wt_hat_beladepos_nicht_verlassen := FALSE;
			sm_tagnummer_ungueltig := FALSE;
			sm_wt_hat_kein_tag := FALSE;
			sm_sensorfehler_beladepos := FALSE;
			sm_tagreader_nicht_fertig := FALSE;
			sm_wt_zu_frueh_in_zelle := FALSE;
			sm_keine_bandfreigabe := FALSE;
			bm_abfrage_wt_auf_beladepos := FALSE;
			bm_warte_anforderung := FALSE;
			bm_warte_auf_wt_an_stopper := FALSE;
			balluff_tag_reader.st_ctrl.in.b_start_lesen := FALSE;
			balluff_tag_reader.st_ctrl.in.b_start_schreiben := FALSE;
			a_station_vorher_out_erlaubnis := FALSE;
			a_station_vorher_out_angekommen := FALSE;
			bMerkerSchrittketteKommtVonInit := TRUE;
		END_IF

		(*-----------------------Weiterschaltbedingungen----------------------------*)
		IF st_ctrl_in.b_init THEN
			zyl_wt_zentrierer_tisch.st_ctrl.in.b_quittieren := FALSE;
			zyl_wt_stopper_tisch.st_ctrl.in.b_quittieren := FALSE;
			zyl_wt_zentrierer_tisch.st_ctrl.in.b_ausfahren := FALSE;
			fb_state_entry.i16_next_step := 20;
		END_IF

(*=======================================================*)
	20: (* Initialisierung: Stopper ausfahren *)
		IF fb_state_entry.E THEN
			zyl_wt_stopper_tisch.st_ctrl.in.b_ausfahren := TRUE;
		END_IF

		(*-----------------------Weiterschaltbedingungen----------------------------*)
		IF zyl_wt_stopper_tisch.st_ctrl.out.b_ausgefahren THEN
			zyl_wt_stopper_tisch.st_ctrl.in.b_ausfahren := FALSE;
			a_station_vorher_out_angekommen := TRUE;	(* benötigtes Signal, damit es an der Vorgängerzelle in "ST_WT_Transport_Abgabe" weiter gehen kann *)
			fb_state_entry.i16_next_step := BEREIT;
		END_IF

(*=======================================================*)
	BEREIT:	(* Warte auf Start von Kontroller *)
		IF fb_state_entry.E THEN
			st_ctrl_out.b_bereit := TRUE;
			st_ctrl_out.b_fertig := TRUE;
			stueckzahlen.st_ctrl.in.b_gutteil_produziert := FALSE;
		END_IF

		(*-----------------------Weiterschaltbedingungen----------------------------*)
		(* WT Transport aktiv oder in Simulation *)
		IF st_config.b_station_aktiv OR st_config.b_station_in_simulation THEN

			IF st_ctrl_in.b_start THEN
			(* WT Transport gestartet *)
				st_ctrl_out.b_fertig := FALSE;
				fb_ton_wz.IN := FALSE;
				st_ctrl_out.b_kontroller_start := TRUE;
				(* Abfrage, ob Schrittkette von Init kommt und ob WT auf Beladepos ist *)
				IF bMerkerSchrittketteKommtVonInit AND
					e_wt_auf_beladepos THEN
					fb_state_entry.i16_next_step := 170;	(* WT auslesen und prüfen, ob dieser schon bestückt wurde *)
				ELSE
					fb_state_entry.i16_next_step := 110;
				END_IF
			END_IF

		(* WT-Transport nicht aktiv  *)
		ELSE
			IF fb_r_trig_start.Q THEN
			(* Nur Z-Achse gestartet *)
				st_ctrl_out.b_fertig := FALSE;
				fb_ton_wz.IN := FALSE;
				fb_state_entry.i16_next_step := 500;
			END_IF
		END_IF

		IF fb_state_entry.X THEN
			bMerkerSchrittketteKommtVonInit := FALSE;
		END_IF

(*=======================================================*)
	105: (* Schreibe Daten auf Tag *)
		IF fb_state_entry.E THEN
			(* WT wird auf jeden Fall mit "nio" beschrieben *)
			ST_Markiere_WT_NIO();
		END_IF

		(*-----------------------Weiterschaltbedingungen----------------------------*)
		IF balluff_tag_reader.st_ctrl.out.b_fertig AND NOT fb_state_entry.E THEN
			balluff_tag_reader.st_ctrl.in.b_start_schreiben := FALSE;
			fb_state_entry.i16_next_step := 110;
		END_IF

